		IF 前左轮力偏差 >200 THEN
			前左轮力偏差 := 200;
		END_IF
		IF 0< 前左轮力偏差 AND 前左轮力偏差 < 150 THEN
			前左轮力偏差 := 0;
		END_IF
		IF 前左轮力偏差 <-200 THEN
			前左轮力偏差 := -200;
		END_IF
		IF -170< 前左轮力偏差 AND 前左轮力偏差 < 0 THEN
			前左轮力偏差 := 0;
		END_IF
		
		IF 前右轮力偏差 >200 THEN
			前右轮力偏差 := 200;
		END_IF
		IF 前右轮力偏差 <-200 THEN
			前右轮力偏差 := -200;
		END_IF
		IF -170< 前右轮力偏差 AND 前右轮力偏差 < 0 THEN
			前右轮力偏差 := 0;
		END_IF
		IF 0< 前右轮力偏差 AND 前右轮力偏差 < 150 THEN
			前右轮力偏差 := 0;
		END_IF

		IF 后左轮力偏差 >200 THEN
			后左轮力偏差 := 200;
		END_IF
		IF 后左轮力偏差 <-200 THEN
			后左轮力偏差 := -200;
		END_IF
		IF -170< 后左轮力偏差 AND 后左轮力偏差 < 0 THEN
			后左轮力偏差 := 0;
		END_IF
		IF 0< 后左轮力偏差 AND 后左轮力偏差 < 150 THEN
			后左轮力偏差 := 0;
		END_IF
		
		IF 后右轮力偏差 >200 THEN
			后右轮力偏差 := 200;
		END_IF
		IF 后右轮力偏差 <-200 THEN
			后右轮力偏差 := -200;
		END_IF
		IF -170< 后右轮力偏差 AND 后右轮力偏差 < 0 THEN
			后右轮力偏差 := 0;
		END_IF
		IF 0< 后右轮力偏差 AND 后右轮力偏差 < 150 THEN
			后右轮力偏差 := 0;
		END_IF
		
		偏差值pitch := -目标值pitch + pitch角度滤波;
		偏差值roll := -目标值roll + roll角度滤波;
		
		PITCH := (pitch角度滤波 - v_pitch)/0.005;
		ROLL := (roll角度滤波 - v_roll)/0.005;

		//角速度滤波
		PITCH滤波 := B0 * PITCH + B1 * PITCH_x1 + B2 * PITCH_x2 - A1 * PITCH_y1 - A2 * PITCH_y2;
		PITCH_x2 := PITCH_x1;
		PITCH_x1 := PITCH;
		PITCH_y2 := PITCH_y1;
		PITCH_y1 := PITCH滤波;
		
		ROLL滤波 := B0 * ROLL + B1 * ROLL_x1 + B2 * ROLL_x2 - A1 * ROLL_y1 - A2 * ROLL_y2;
		ROLL_x2 := ROLL_x1;
		ROLL_x1 := ROLL;
		ROLL_y2 := ROLL_y1;
		ROLL_y1 := ROLL滤波;
		
// 死区处理
		IF ABS(偏差值pitch) < 误差死区 THEN 偏差值pitch := 0.0; END_IF;
		IF ABS(偏差值roll) < 误差死区 THEN 偏差值roll := 0.0; END_IF;
		
		IF ABS(偏差值pitch) < 误差死区 THEN PITCH滤波 := 0.0; END_IF;
		IF ABS(偏差值roll) < 误差死区 THEN ROLL滤波 := 0.0; END_IF;

		KP_roll := 0.45;
		KD_roll := 0.3;
		KI_roll := 0.0045;
		KP_pitch := 0.75;
		KD_pitch := 0.55;
		KI_pitch := 0.0045;

		//记录数据
		KD数据pitch := 偏差值pitch - 2*e_pitch_prev1 + e_pitch_prev2;
		KP数据pitch := 偏差值pitch - e_pitch_prev1;
		KI数据pitch := 偏差值pitch;
		KD数据roll := 偏差值roll - 2*e_roll_prev1 + e_roll_prev2;
		KP数据roll := 偏差值roll - e_roll_prev1;
		KI数据roll := 偏差值roll;
		
		// KP_pitch滤波计算
		KP数据pitch滤波 := B0 * KP数据pitch + B1 * KP_pitch_x1 + B2 * KP_pitch_x2 - A1 * KP_pitch_y1 - A2 * KP_pitch_y2;
		KP_pitch_x2 := KP_pitch_x1;
		KP_pitch_x1 := KP数据pitch;
		KP_pitch_y2 := KP_pitch_y1;
		KP_pitch_y1 := KP数据pitch滤波;
		
		KD数据pitch滤波 := B0 * KD数据pitch + B1 * KD_pitch_x1 + B2 * KD_pitch_x2 - A1 * KD_pitch_y1 - A2 * KD_pitch_y2;
		KD_pitch_x2 := KD_pitch_x1;
		KD_pitch_x1 := KD数据pitch;
		KD_pitch_y2 := KD_pitch_y1;
		KD_pitch_y1 := KD数据pitch滤波;
		
		KP数据roll滤波 := B0 * KP数据roll + B1 * KP_roll_x1 + B2 * KP_roll_x2 - A1 * KP_roll_y1 - A2 * KP_roll_y2;
		KP_roll_x2 := KP_roll_x1;
		KP_roll_x1 := KP数据roll;
		KP_roll_y2 := KP_roll_y1;
		KP_roll_y1 := KP数据roll滤波;

		KD数据roll滤波 := B0 * KD数据roll + B1 * KD_roll_x1 + B2 * KD_roll_x2 - A1 * KD_roll_y1 - A2 * KD_roll_y2;
		KD_roll_x2 := KD_roll_x1;
		KD_roll_x1 := KD数据roll;
		KD_roll_y2 := KD_roll_y1;
		KD_roll_y1 := KD数据roll滤波;

// PID输出
		控制量pitch := KP_pitch * (KP数据pitch滤波) 
            + KI_pitch * 偏差值pitch 
            + KD_pitch * (KD数据pitch滤波);
		
		控制量roll := KP_roll * (KP数据roll滤波) 
           + KI_roll * 偏差值roll 
           + KD_roll * (KD数据roll滤波);
		
		v_pitch := pitch角度滤波;
		v_roll := roll角度滤波;
		
		前左轮date_l := +控制量pitch - 控制量roll;
		前右轮date_l := +控制量pitch + 控制量roll;
		后左轮date_l := -控制量pitch - 控制量roll;
		后右轮date_l := -控制量pitch + 控制量roll;
		
		// 更新历史误差
		e_pitch_prev2 := e_pitch_prev1;
		e_pitch_prev1 := 偏差值pitch;
		e_roll_prev2 := e_roll_prev1;
		e_roll_prev1 := 偏差值roll;
        
		
		//弃用的力增益分段式		
		// 		IF ABS(前左轮力偏差)>180 THEN
		// 			KP_force前左 := 0.0012;
		// 			ELSE
		// 			KP_force前左 := 0.0006;
		// 		END_IF
		// 		
		// 		IF ABS(前右轮力偏差)>180 THEN
		// 			KP_force前右 := 0.0012;
		// 			ELSE
		// 			KP_force前右 := 0.0006;
		// 		END_IF
		// 
		// 		IF ABS(后左轮力偏差)>180 THEN
		// 			KP_force后左 := 0.0012;
		// 			ELSE
		// 			KP_force后左 := 0.0006;
		// 		END_IF
		// 
		// 		IF ABS(后右轮力偏差)>180 THEN
		// 			KP_force后右 := 0.0012;
		// 			ELSE
		// 			KP_force后右 := 0.0006;
		// 		END_IF

//调节力的增益与加速度
		// 前左轮速度滤波计算
		前左轮速度滤波 := B0 * 前左轮行驶速度 + B1 * FLa_x1 + B2 * FLa_x2 - A1 * FLa_y1 - A2 * FLa_y2;
		FLa_x2 := FLa_x1;
		FLa_x1 := 前左轮行驶速度;
		FLa_y2 := FLa_y1;
		FLa_y1 := 前左轮速度滤波;
		
		// 前右------------------------
		前右轮速度滤波 := B0 * 前右轮行驶速度 + B1 * FRa_x1 + B2 * FRa_x2 - A1 * FRa_y1 - A2 * FRa_y2;
		FRa_x2 := FRa_x1;
		FRa_x1 := 前右轮行驶速度;
		FRa_y2 := FRa_y1;
		FRa_y1 := 前右轮速度滤波;
		
		// 后左------------------------
		后左轮速度滤波 := B0 * 后左轮行驶速度 + B1 * RLa_x1 + B2 * RLa_x2 - A1 * RLa_y1 - A2 * RLa_y2;
		RLa_x2 := RLa_x1;
		RLa_x1 := 后左轮行驶速度;
		RLa_y2 := RLa_y1;
		RLa_y1 := 后左轮速度滤波;
		
		// 后右------------------------
		后右轮速度滤波 := B0 * 后右轮行驶速度 + B1 * RRa_x1 + B2 * RRa_x2 - A1 * RRa_y1 - A2 * RRa_y2;
		RRa_x2 := RRa_x1;
		RRa_x1 := 后右轮行驶速度;
		RRa_y2 := RRa_y1;
		RRa_y1 := 后右轮速度滤波;

        前左轮加速度滤波 := (前左轮速度滤波 - 前左轮速度滤波L)/0.005;
		前右轮加速度滤波 := (前右轮速度滤波 - 前右轮速度滤波L)/0.005;
		后左轮加速度滤波 := (后左轮速度滤波 - 后左轮速度滤波L)/0.005;
		后右轮加速度滤波 := (后右轮速度滤波 - 后右轮速度滤波L)/0.005;
		
		前左轮速度滤波L := 前左轮速度滤波;
		前右轮速度滤波L := 前右轮速度滤波;
		后左轮速度滤波L := 后左轮速度滤波;
		后右轮速度滤波L := 后右轮速度滤波;

// 弃用的定时器
		//accel_high := (ABS(后左轮加速度滤波) >= 150);
		//// 配置并运行定时器（预设时间50ms）
		//timer_high(IN:=accel_high, PT:=T#50MS);
		//IF timer_high.Q THEN
		//KP_force后左 :=  150*KP_force后左/ABS(后左轮加速度滤波) ;
		//KP_force前左 :=  150*KP_force前左/ABS(后左轮加速度滤波) ;
		//KP_force前右 :=  150*KP_force前右/ABS(后左轮加速度滤波) ;
		//KP_force后右 :=  150*KP_force后右/ABS(后左轮加速度滤波) ;
		//END_IF

		// 后左轮加速度计数器
		IF ABS(后左轮加速度滤波) >= 200 THEN
			a轮与kp力计数器 := a轮与kp力计数器 + 1;
		ELSE
			a轮与kp力计数器 := 0;
		END_IF;
		
		// 前左轮KP_force自适应调整
		IF ABS(前左轮力偏差) > 180 THEN
			KP_force前左 := KP_force前左 + 0.000011;
			IF KP_force前左 >= 0.0003 THEN
				KP_force前左 := 0.0003;
			END_IF;	
		ELSIF a轮与kp力计数器 >= 10 THEN
			KP_force前左 := KP_force前左 - 0.000011;
			IF KP_force前左 <= 0 THEN
				KP_force前左 := 0;
			END_IF;
		ELSIF a轮与kp力计数器 = 0 THEN
			IF KP_force前左 < 0.00015 THEN
				KP_force前左 := KP_force前左 + 0.000012;
			ELSIF KP_force前左 > 0.00015 THEN
				KP_force前左 := KP_force前左 - 0.000012;
			END_IF;
		END_IF;

		// 前右轮KP_force自适应调整
		IF ABS(前右轮力偏差) > 180 THEN
			KP_force前右 := KP_force前右 + 0.000011;
			IF KP_force前右 >= 0.0003 THEN
				KP_force前右 := 0.0003;
			END_IF;	
		ELSIF a轮与kp力计数器 >= 10 THEN
			KP_force前右 := KP_force前右 - 0.000011;
			IF KP_force前右 <= 0 THEN
				KP_force前右 := 0;
			END_IF;
		ELSIF a轮与kp力计数器 = 0 THEN
			IF KP_force前右 < 0.00015 THEN
				KP_force前右 := KP_force前右 + 0.000012;
			ELSIF KP_force前右 > 0.00015 THEN
				KP_force前右 := KP_force前右 - 0.000012;
			END_IF;
		END_IF;

		// 后左轮KP_force自适应调整
		IF ABS(后左轮力偏差) > 180 THEN
			KP_force后左 := KP_force后左 + 0.000012;
			IF KP_force后左 >= 0.0003 THEN
				KP_force后左 := 0.0003;
			END_IF;	
		ELSIF a轮与kp力计数器 >= 10 THEN
			KP_force后左 := KP_force后左 - 0.000012;
			IF KP_force后左 <= 0 THEN
				KP_force后左 := 0;
			END_IF;
		ELSIF a轮与kp力计数器 = 0 THEN
			IF KP_force后左 < 0.00015 THEN
				KP_force后左 := KP_force后左 + 0.000012;
			ELSIF KP_force后左 > 0.00015 THEN
				KP_force后左 := KP_force后左 - 0.000012;
			END_IF;
		END_IF;

		// 后右轮KP_force自适应调整
		IF ABS(后右轮力偏差) > 180 THEN
			KP_force后右 := KP_force后右 + 0.000012;
			IF KP_force后右 >= 0.0003 THEN
				KP_force后右 := 0.0003;
			END_IF;	
		ELSIF a轮与kp力计数器 >= 10 THEN
			KP_force后右 := KP_force后右 - 0.000012;
			IF KP_force后右 <= 0 THEN
				KP_force后右 := 0;
			END_IF;
		ELSIF a轮与kp力计数器 = 0 THEN
			IF KP_force后右 < 0.00015 THEN
				KP_force后右 := KP_force后右 + 0.000012;
			ELSIF KP_force后右 > 0.00015 THEN
				KP_force后右 := KP_force后右 - 0.000012;
			END_IF;
		END_IF;

		// 		IF ABS(后左轮加速度滤波) >= 200 THEN
		// 			KP_force后左 := 0;
		// 			KP_force前左 := 0;
		// 			KP_force前右 := 0;
		// 			KP_force后右 := 0;
		// 			ELSIF ABS(后左轮加速度滤波) >= 20 THEN
		// 			KP_force后左 :=  20*KP_force后左/ABS(后左轮加速度滤波) ;
		// 			KP_force前左 :=  20*KP_force前左/ABS(后左轮加速度滤波) ;
		// 			KP_force前右 :=  20*KP_force前右/ABS(后左轮加速度滤波) ;
		// 			KP_force后右 :=  20*KP_force后右/ABS(后左轮加速度滤波) ;
		// 		END_IF
		
		前左轮date := (前左轮date_l - (前左轮力偏差 * KP_force前左));
		前右轮date := (前右轮date_l - (前右轮力偏差 * KP_force前右));
		后左轮date := (后左轮date_l - (后左轮力偏差 * KP_force后左));
		后右轮date := (后右轮date_l - (后右轮力偏差 * KP_force后右));
		
		前左轮date_F := 前左轮力偏差 * KP_force前左;
		前右轮date_F := 前右轮力偏差 * KP_force前右;
		后左轮date_F := 后左轮力偏差 * KP_force后左;
		后右轮date_F := 后右轮力偏差 * KP_force后右;
		
		// 计算预期位置
		前左轮new := (前左轮输出 + 前左轮date);
		前右轮new := (前右轮输出 + 前右轮date);
		后左轮new := (后左轮输出 + 后左轮date);
		后右轮new := (后右轮输出 + 后右轮date);
		
//执行器极限补偿
		//前轮组极限检查
		前轮组上极限 := (前左轮new >= 执行器行程限制) AND (前右轮new >= 执行器行程限制);
		前轮组下极限 := (前左轮new <= -执行器行程限制) AND (前右轮new <= -执行器行程限制);
		
		// 后轮组极限检查
		后轮组上极限 := (后左轮new >= 执行器行程限制) AND (后右轮new >= 执行器行程限制);
		后轮组下极限 := (后左轮new <= -执行器行程限制) AND (后右轮new <= -执行器行程限制);
		
		// Pitch轴补偿
		IF 前轮组上极限 AND (偏差值pitch > 误差死区) THEN
			后左轮date := 后左轮date - 最大调整速度 * 0.01;
			后右轮date := 后右轮date - 最大调整速度 * 0.01;
		ELSIF 前轮组下极限 AND (偏差值pitch < -误差死区) THEN
			后左轮date := 后左轮date + 最大调整速度 * 0.01;
			后右轮date := 后右轮date + 最大调整速度 * 0.01;
		END_IF;
		
		IF 后轮组上极限 AND (偏差值pitch < -误差死区) THEN
			前左轮date := 前左轮date + 最大调整速度 * 0.01;
			前右轮date := 前右轮date + 最大调整速度 * 0.01;
		ELSIF 后轮组下极限 AND (偏差值pitch > 误差死区) THEN
			前左轮date := 前左轮date - 最大调整速度 * 0.01;
			前右轮date := 前右轮date - 最大调整速度 * 0.01;
		END_IF;
		
		// 左侧极限检查
		左组轮上极限 := (前左轮new >= 执行器行程限制) AND (后左轮new >= 执行器行程限制);
		左组轮下极限 := (前左轮new <= -执行器行程限制) AND (后左轮new <= -执行器行程限制);
		
		// 右侧极限检查
		右组轮上极限 := (前右轮date >= 执行器行程限制) AND (后右轮date >= 执行器行程限制);
		右组轮下极限 := (前右轮date <= -执行器行程限制) AND (后右轮date <= -执行器行程限制);
		
		IF 左组轮上极限 AND (偏差值roll > 误差死区) THEN
			前右轮date := 前右轮date - 最大调整速度 * 0.01;
			后右轮date := 后右轮date - 最大调整速度 * 0.01;
		ELSIF 左组轮下极限 AND (偏差值roll < -误差死区) THEN
			前右轮date := 前右轮date + 最大调整速度 * 0.01;
			后右轮date := 后右轮date + 最大调整速度 * 0.01;
		END_IF;
		
		IF 右组轮上极限 AND (偏差值roll < -误差死区) THEN
			前左轮date := 前左轮date - 最大调整速度 * 0.01;
			后左轮date := 后左轮date - 最大调整速度 * 0.01;
		ELSIF 右组轮下极限 AND (偏差值roll > 误差死区) THEN
			前左轮date := 前左轮date + 最大调整速度 * 0.01;
			后左轮date := 后左轮date + 最大调整速度 * 0.01;
		END_IF;
		
		//最终限幅及输出
		// 速度限幅
		前左轮date := LIMIT(前左轮date, -最大调整速度, 最大调整速度);
		前右轮date := LIMIT(前右轮date, -最大调整速度, 最大调整速度);
		后左轮date := LIMIT(后左轮date, -最大调整速度, 最大调整速度);
		后右轮date := LIMIT(后右轮date, -最大调整速度, 最大调整速度);

//弃用的速度控制
		// 前左轮速度计算
		IF ABS(前左轮date) > 10.0 THEN
			前左轮速度 := 50.0;
		ELSIF ABS(前左轮date) < 0.05 THEN
			前左轮速度 := 0.0;
		ELSE
			前左轮速度 := (前左轮date) * (50.0 / 10);  // 100/(10.0-0.5)=10.5263
		END_IF;
		
		// 前右轮速度计算
		IF ABS(前右轮date) > 10.0 THEN
			前右轮速度 := 50.0;
		ELSIF ABS(前右轮date) < 0.05 THEN
			前右轮速度 := 0.0;
		ELSE
			前右轮速度 := (前右轮date) * (50.0 / 10);
		END_IF;
		
		// 后左轮速度计算
		IF ABS(后左轮date) > 10.0 THEN
			后左轮速度 := 50.0;
		ELSIF ABS(后左轮date) < 0.05 THEN
			后左轮速度 := 0.0;
		ELSE
			后左轮速度 := (后左轮date) * (50.0 / 10);
		END_IF;
		
		// 后右轮速度计算
		IF ABS(后右轮date) > 10.0 THEN
			后右轮速度 := 50.0;
		ELSIF ABS(后右轮date) < 0.05 THEN
			后右轮速度 := 0.0;
		ELSE
			后右轮速度 := (后右轮date) * (50.0 / 10);
		END_IF;
		
		delta前左 := 前左轮date - 前左轮date_l_prev;
		delta前右 := 前右轮date - 前右轮date_l_prev;
		delta后左 := 后左轮date - 后左轮date_l_prev;
		delta后右 := 后右轮date - 后右轮date_l_prev;
		
		//前左轮date_prev := 前左轮date;
		//前右轮date_prev := 前右轮date;
		//后左轮date_prev := 后左轮date;
		//后右轮date_prev := 后右轮date;

//轮date增幅限制
		//前左
		IF delta前左 > 0 THEN
			sign := 1;      // 正方向
		ELSIF delta前左 < 0 THEN
			sign := -1;     // 负方向
		ELSE
			sign := 0;      // 无变化
		END_IF;
		
		IF ABS(delta前左) > delta_threshold THEN
			// 超过阈值时，按符号限幅
			前左轮date := 前左轮date_l_prev + (sign * delta_threshold);
		END_IF;
		//前右
		IF delta前右 > 0 THEN
			sign := 1;      // 正方向
		ELSIF delta前右 < 0 THEN
			sign := -1;     // 负方向
		ELSE
			sign := 0;      // 无变化
		END_IF;
		
		IF ABS(delta前右) > delta_threshold THEN
			// 超过阈值时，按符号限幅
			前右轮date := 前右轮date_l_prev + (sign * delta_threshold);
		END_IF;
        //后左
		IF delta后左 > 0 THEN
			sign := 1;      // 正方向
		ELSIF delta后左 < 0 THEN
			sign := -1;     // 负方向
		ELSE
			sign := 0;      // 无变化
		END_IF;
		
		IF ABS(delta后左) > delta_threshold THEN
			// 超过阈值时，按符号限幅
			后左轮date := 后左轮date_l_prev + (sign * delta_threshold);
		END_IF;
		//后右
		IF delta后右 > 0 THEN
			sign := 1;      // 正方向
		ELSIF delta后右 < 0 THEN
			sign := -1;     // 负方向
		ELSE
			sign := 0;      // 无变化
		END_IF;
		
		IF ABS(delta后右) > delta_threshold THEN
			// 超过阈值时，按符号限幅
			后右轮date := 后右轮date_l_prev + (sign * delta_threshold);
		END_IF;

		前左轮date_l_prev := 前左轮date;
		前右轮date_l_prev := 前右轮date;
		后右轮date_l_prev := 后右轮date;
		后左轮date_l_prev := 后左轮date;

//轮date滤波
		// 前左轮滤波计算
		// ----------------------------
		前左轮date滤波 := B0 * 前左轮date + B1 * FLdate_x1 + B2 * FLdate_x2 - A1 * FLdate_y1 - A2 * FLdate_y2;
		// 更新状态
		FLdate_x2 := FLdate_x1;
		FLdate_x1 := 前左轮date;
		FLdate_y2 := FLdate_y1;
		FLdate_y1 := 前左轮date滤波;
		
		// ----------------------------
		// 前右轮滤波计算
		// ----------------------------
		前右轮date滤波 := B0 * 前右轮date + B1 * FRdate_x1 + B2 * FRdate_x2 - A1 * FRdate_y1 - A2 * FRdate_y2;
		// 更新状态
		FRdate_x2 := FRdate_x1;
		FRdate_x1 := 前右轮date;
		FRdate_y2 := FRdate_y1;
		FRdate_y1 := 前右轮date滤波;
		
		// ----------------------------
		// 后左轮滤波计算
		// ----------------------------
		后左轮date滤波 := B0 * 后左轮date + B1 * BLdate_x1 + B2 * BLdate_x2 - A1 * BLdate_y1 - A2 * BLdate_y2;
		// 更新状态
		BLdate_x2 := BLdate_x1;
		BLdate_x1 := 后左轮date;
		BLdate_y2 := BLdate_y1;
		BLdate_y1 := 后左轮date滤波;
		
		// ----------------------------
		// 后右轮滤波计算
		// ----------------------------
		后右轮date滤波 := B0 * 后右轮date + B1 * BRdate_x1 + B2 * BRdate_x2 - A1 * BRdate_y1 - A2 * BRdate_y2;
		// 更新状态
		BRdate_x2 := BRdate_x1;
		BRdate_x1 := 后右轮date;
		BRdate_y2 := BRdate_y1;
		BRdate_y1 := 后右轮date滤波;

// 前左轮date滤波应用限幅（±0.01米）
		// 前左轮date滤波 := LIMIT(前左轮date滤波, -0.25, 0.25);
		// 前右轮date滤波 := LIMIT(前右轮date滤波, -0.25, 0.25);
		// 后左轮date滤波 := LIMIT(后左轮date滤波, -0.25, 0.25);
		// 后右轮date滤波 := LIMIT(后右轮date滤波, -0.25, 0.25);

		平均实际长度 := (前左轮实际长度 + 前右轮实际长度 + 后左轮实际长度 + 后右轮实际长度) / 4.0;

		IF 平均实际长度>0.5 AND ABS(pitch角度滤波) < 0.5 AND ABS(roll角度滤波) < 0.5 THEN
			// 模式A：偏差均小时，用比例调整输出
			前左轮输出 := LIMIT(前左轮输出 + 前左轮date滤波 + 前左轮调整量滤波 - kp * 15, -执行器行程限制, 执行器行程限制);
			前右轮输出 := LIMIT(前右轮输出 + 前右轮date滤波 + 前右轮调整量滤波 - kp * 15, -执行器行程限制, 执行器行程限制);
			后左轮输出 := LIMIT(后左轮输出 + 后左轮date滤波 + 后左轮调整量滤波 - kp * 15, -执行器行程限制, 执行器行程限制);
			后右轮输出 := LIMIT(后右轮实际长度 + 后右轮date滤波 + 后右轮调整量滤波 - kp * 15, -执行器行程限制, 执行器行程限制);
			ELSE IF 平均实际长度<-0.5 AND ABS(pitch角度滤波) < 0.5 AND ABS(roll角度滤波) < 0.5 THEN
			前左轮输出 := LIMIT(前左轮输出 + 前左轮date滤波 + 前左轮调整量滤波 + kp * 15, -执行器行程限制, 执行器行程限制);
			前右轮输出 := LIMIT(前右轮输出 + 前右轮date滤波 + 前右轮调整量滤波 + kp * 15, -执行器行程限制, 执行器行程限制);
			后左轮输出 := LIMIT(后左轮输出 + 后左轮date滤波 + 后左轮调整量滤波 + kp * 15, -执行器行程限制, 执行器行程限制);
			后右轮输出 := LIMIT(后右轮输出 + 后右轮date滤波 + 后右轮调整量滤波 + kp * 15, -执行器行程限制, 执行器行程限制);
					ELSE
						前左轮输出 := LIMIT(前左轮输出 + 前左轮date滤波 + 前左轮调整量滤波, -执行器行程限制, 执行器行程限制);
						前右轮输出 := LIMIT(前右轮输出 + 前右轮date滤波 + 前右轮调整量滤波, -执行器行程限制, 执行器行程限制);
						后左轮输出 := LIMIT(后左轮输出 + 后左轮date滤波 + 后左轮调整量滤波, -执行器行程限制, 执行器行程限制);
						后右轮输出 := LIMIT(后右轮输出 + 后右轮date滤波 + 后右轮调整量滤波, -执行器行程限制, 执行器行程限制);
			     END_IF
		END_IF;

END_FUNCTION_BLOCK

// Device/Application/函数/运动控制/伺服控制
FUNCTION_BLOCK 伺服控制
VAR_INPUT
	pAxis      	: POINTER TO AXIS_REF_SM3;	//定义轴
END_VAR
VAR_OUTPUT
END_VAR
VAR
	前进					: BOOL := FALSE;
	后退					: BOOL := FALSE;
	运动到点开始,运动到点开始1			: BOOL := FALSE;
	相对运动到点开始        : BOOL := FALSE;
	连续运动到点开始        : BOOL := FALSE;
	速度运动到点开始,速度运动到点开始1        : BOOL := FALSE;
	力矩模式切换: BOOL;
	力矩控制,力矩控制1:BOOL;
	暂停        : BOOL := FALSE;
	停止控制    : BOOL := FALSE;
	
	到点位置				: LREAL := 0.0;
	pMC_Jog    			: MC_Jog;
	pMC_Power  			: MC_Power;
	pMC_Reset  			: MC_Reset;
	pMC_MoveAbsolute1,pMC_MoveAbsolute 	: MC_MoveAbsolute;
	pMC_MoveRelative 	: MC_MoveRelative;
	pMC_MoveAdditive    : MC_MoveAdditive;
	pMC_MoveVelocity,pMC_MoveVelocity1    : MC_MoveVelocity;
	pSMC_SetTorque,pSMC_SetTorque1      : SMC_SetTorque;
	pSMC_MoveContinuousAbsolute: SMC_MoveContinuousAbsolute;
	pSMC_SetControllerMode:SMC_SetControllerMode;
	pMC_Halt:MC_Halt;
	pMC_Stop:MC_Stop;
	pSMC3_ReinitDrive:SMC3_ReinitDrive;
	运行速度		: LREAL ;
	运行方向		: INT ;
	
END_VAR
VAR_IN_OUT
	伺服参数    			: 伺服参数结构体;
END_VAR

IF 轴报警=FALSE THEN
CASE 伺服参数.运行模式 OF
	0 :	// 无运动
		前进 := FALSE;
		后退 := FALSE;
		运动到点开始:=FALSE;
		运动到点开始1:=FALSE;
		相对运动到点开始:=FALSE;
		连续运动到点开始:=FALSE;
		速度运动到点开始:=FALSE;
		速度运动到点开始1:=FALSE;
		力矩控制:=FALSE;
		力矩控制1:=FALSE;
		暂停:=FALSE;
		停止控制:=FALSE;
		力矩模式切换:=FALSE;
		//轴复位:=FALSE;
		//轴初始化:=FALSE;
	1 : // 点动运行
		IF 伺服参数.运行方向=TRUE THEN
			前进 := TRUE;
			后退 := FALSE;
		ELSE
			前进 := FALSE;
			后退 := TRUE;
		END_IF
	2 : // 运动到点1
	    运动到点开始1:=FALSE;
		运动到点开始:=TRUE;
	3 : // 相对运动
	    运动到点开始:=FALSE;
		运动到点开始1:=FALSE;
		相对运动到点开始:=TRUE;
		
	4 : // 运动到点2
	    运动到点开始:=FALSE;
		运动到点开始1:=TRUE;
	
    5:
	    暂停:=TRUE;
	6://速度控制1
	    速度运动到点开始1:=FALSE;
	    速度运动到点开始:=TRUE;
		暂停:=FALSE;
	7://速度控制2
	    速度运动到点开始:=FALSE;
	    速度运动到点开始1:=TRUE;
		暂停:=FALSE;
	8://力矩控制1
	    力矩控制1:=FALSE;
		力矩控制:=TRUE;
	9://力矩控制2
	    力矩控制:=FALSE;
		力矩控制1:=TRUE;
	10://停止
	    停止控制:=TRUE;
	11://力矩切换
	    力矩模式切换:=TRUE;
	//12://位置模式
	(*
	13://复位
	    轴复位:=TRUE;
	14://初始化
	    轴初始化:=TRUE;
	*)
END_CASE
END_IF
pMC_Power(
	Axis:= pAxis^,
	Enable:= TRUE,
	bRegulatorOn:= 伺服参数.使能,
	bDriveStart:= TRUE,
	Status=> , 
	bRegulatorRealState=> 伺服参数.使能状态.DONE, 
	bDriveStartRealState=> , 
	Busy=> 伺服参数.使能状态.BUSY, 
	Error=> 伺服参数.使能状态.Error, 
	ErrorID=> 伺服参数.使能状态.ErrorID);

pMC_Jog(
	Axis:= pAxis^,
	JogForward:= 前进,
	JogBackward:= 后退,
	Velocity:= 伺服参数.运行速度,
	Acceleration:= 10000,
	Deceleration:= 10000,
	Jerk:=100000,
	Busy=> 伺服参数.点动运行中,
	CommandAborted=>,
	Error=>, 
	ErrorId=> );

pMC_MoveAbsolute(
	Axis:=pAxis^ , 
	Execute:= 运动到点开始, 
	Position:= 伺服参数.运行位置, 
	Velocity:= 伺服参数.运行速度, 
	Acceleration:= 10000, 
	Deceleration:= 10000, 
	Jerk:= 100000, 
	Direction:= , 
	BufferMode:= 0, 
	Done=> 伺服参数.绝对定位状态.DONE, 
	Busy=> 伺服参数.绝对定位状态.BUSY, 
	CommandAborted=> 伺服参数.绝对定位状态.CommandAborted, 
	Error=> 伺服参数.绝对定位状态.Error, 
	ErrorID=> 伺服参数.绝对定位状态.ErrorID);	

pMC_MoveAbsolute1(
	Axis:=pAxis^ , 
	Execute:= 运动到点开始1, 
	Position:= 伺服参数.运行位置1, 
	Velocity:= 伺服参数.运行速度, 
	Acceleration:= 10000, 
	Deceleration:= 10000, 
	Jerk:= 100000, 
	Direction:= , 
	BufferMode:= 0, 
	Done=> 伺服参数.绝对定位状态1.DONE, 
	Busy=> 伺服参数.绝对定位状态1.BUSY, 
	CommandAborted=> 伺服参数.绝对定位状态1.CommandAborted, 
	Error=> 伺服参数.绝对定位状态1.Error, 
	ErrorID=> 伺服参数.绝对定位状态1.ErrorID);	

pMC_MoveRelative(
	Axis:= pAxis^, 
	Execute:= 相对运动到点开始, 
	Distance:= 伺服参数.运行位置, 
	Velocity:= 伺服参数.运行速度, 
	Acceleration:= 500, 
	Deceleration:= 500, 
	Jerk:= 5000, 
	BufferMode:= 5, 
	Done=> 伺服参数.相对定位状态.DONE, 
	Busy=> 伺服参数.相对定位状态.BUSY, 
	Active=> , 
	CommandAborted=> 伺服参数.相对定位状态.CommandAborted, 
	Error=> 伺服参数.相对定位状态.Error, 
	ErrorID=> 伺服参数.相对定位状态.ErrorID);
(*
pMC_MoveAdditive(
	Axis:= pAxis^, 
	Execute:= 运动到点开始1, 
	Distance:= 伺服参数.运行位置1, 
	Velocity:= 伺服参数.运行速度, 
	Acceleration:= 5000, 
	Deceleration:= 5000, 
	Jerk:= 50000, 
	Done=> 伺服参数.运动到点完成1, 
	Busy=> , 
	CommandAborted=> , 
	Error=> , 
	ErrorID=> );
*)
(*
pSMC_MoveContinuousAbsolute(
	Axis:= pAxis^, 
	Execute:= 连续运动到点开始, 
	Position:= 伺服参数.运行位置, 
	Velocity:= 伺服参数.运行速度, 
	EndVelocity:=伺服参数.结束运行速度, 
	EndVelocityDirection:= , 
	Acceleration:= 500, 
	Deceleration:= 500, 
	Jerk:= 5000, 
	Direction:= , 
	AdaptEndVelToAvoidOvershoot:=TRUE,
	InEndVelocity=> , 
	PositionReached=> 伺服参数.连续运动到点完成, 
	Busy=> , 
	CommandAborted=> , 
	Error=> , 
	ErrorID=> );
*)
pMC_Halt(
	Axis:= pAxis^, 
	Execute:= 暂停, 
	Deceleration:= 500, 
	Jerk:= 5000, 
	Done=> 伺服参数.暂停状态.DONE, 
	Busy=> 伺服参数.暂停状态.BUSY, 
	CommandAborted=> 伺服参数.暂停状态.CommandAborted, 
	Error=> 伺服参数.暂停状态.Error, 
	ErrorID=> 伺服参数.暂停状态.ErrorID);
	
pMC_Reset(
	Axis:= pAxis^, 
	Execute:= 伺服参数.轴复位, 
	Done=> 伺服参数.复位状态.DONE, 
	Busy=> 伺服参数.复位状态.BUSY, 
	Error=> 伺服参数.复位状态.Error, 
	ErrorID=> 伺服参数.复位状态.ErrorID);
pSMC3_ReinitDrive(
	Axis:= pAxis^, 
	bExecute:= 伺服参数.轴初始化, 
	bVirtual:= , 
	bDone=> 伺服参数.初始化状态.DONE, 
	bBusy=> 伺服参数.初始化状态.BUSY, 
	bError=> 伺服参数.初始化状态.Error, 
	nErrorID=> 伺服参数.初始化状态.ErrorID);


////////////////////////////////////////////////////////////////////////////////////////////////////////

pMC_MoveVelocity(
	Axis:= pAxis^, 
	Execute:= 速度运动到点开始 , 
	Velocity:= 伺服参数.运行控制速度, 
	Acceleration:= 200, 
	Deceleration:= 300, 
	Jerk:= 200, 
	Direction:= 伺服参数.运行控制方向, 
	BufferMode:= , 
	InVelocity=> 伺服参数.速度运动状态.DONE, 
	Busy=> 伺服参数.速度运动状态.BUSY, 
	Active=> , 
	CommandAborted=> 伺服参数.速度运动状态.CommandAborted, 
	Error=> 伺服参数.速度运动状态.Error, 
	ErrorID=> 伺服参数.速度运动状态.ErrorID);
	
pMC_MoveVelocity1(
	Axis:= pAxis^, 
	Execute:= 速度运动到点开始1 , 
	Velocity:= 伺服参数.运行控制速度1, 
	Acceleration:= 200, 
	Deceleration:= 300, 
	Jerk:= 200, 
	Direction:= 伺服参数.运行控制方向, 
	BufferMode:= , 
	InVelocity=> 伺服参数.速度运动状态1.DONE, 
	Busy=> 伺服参数.速度运动状态1.BUSY, 
	Active=> , 
	CommandAborted=> 伺服参数.速度运动状态1.CommandAborted, 
	Error=> 伺服参数.速度运动状态1.Error, 
	ErrorID=> 伺服参数.速度运动状态1.ErrorID);
//轴程序控制.伺服反馈_速度运行_done := 速度运动状态.DONE;	

pSMC_SetControllerMode(
	Axis:= pAxis^, 
	bExecute:= 力矩模式切换 AND NOT (pAxis^.nAxisState = 1 OR pAxis^.nAxisState = 2 OR pAxis^.nAxisState = 7), 
	nControllerMode:= 伺服参数.控制模式, 
	bDone=> 伺服参数.控制模式切换状态.DONE, 
	bBusy=> 伺服参数.控制模式切换状态.BUSY, 
	bError=> 伺服参数.控制模式切换状态.Error, 
	nErrorID=> 伺服参数.控制模式切换状态.ErrorID);
//伺服参数.控制模式切换完成 := pSMC_SetControllerMode.bDone; 



pSMC_SetTorque(
	Axis:=pAxis^ ,
	bEnable:=力矩控制 AND 伺服参数.控制模式 = SMC_torque  ,
	fTorque:=伺服参数.设定力矩 ,
    bBusy => , 
    bError => , 
    nErrorID => , 
	bBusy=> );
	
pSMC_SetTorque1(
	Axis:=pAxis^ ,
	bEnable:=力矩控制1 AND 伺服参数.控制模式 = SMC_torque  ,
	fTorque:=伺服参数.设定力矩1 ,
    bBusy => , 
    bError => , 
    nErrorID => , 
	bBusy=> );
//轴程序控制.伺服反馈_力矩运行_done := 力矩运动状态.BUSY;

pMC_Stop(
	Axis:= pAxis^, 
	Execute:= 伺服参数.停止控制, 
	Deceleration:= 2000, 
	Jerk:= 20000, 
	Done=> 伺服参数.停止状态.DONE, 
	Busy=> 伺服参数.停止状态.BUSY, 
	Error=> 伺服参数.停止状态.Error, 
	ErrorID=> 伺服参数.停止状态.ErrorID);
//轴程序控制.伺服反馈_停止_done := 停止状态.DONE;




伺服参数.指令位置 := pAxis^.fSetPosition;
伺服参数.指令力矩 := pAxis^.fSetTorque;
伺服参数.指令速度 := pAxis^.fSetVelocity;
伺服参数.反馈位置 := pAxis^.fActPosition;
伺服参数.反馈力矩 := pAxis^.fActTorque;
伺服参数.反馈速度 := pAxis^.fActVelocity;
伺服参数.反馈电流 := pAxis^.fActCurrent;
伺服参数.反馈状态 := pAxis^.nAxisState;

END_FUNCTION_BLOCK

// Device/Application/末端控制
PROGRAM 末端控制
VAR
	末端碰撞调整开关	: BOOL := FALSE;
	末端速度			: LREAL := 100.0;
	伸缩轴伺服控制    : 伺服控制;
	上卷扬伺服控制    : 伺服控制;
	下卷扬伺服控制    : 伺服控制;
	滚刷伺服控制    	: 伺服控制;
	
	// 滤波参数
	滤波系数			: LREAL := 0.1;
	上卷扬滤波力矩	: LREAL;
	下卷扬滤波力矩	: LREAL;
	上卷扬上周期力矩	: LREAL;
	下卷扬上周期力矩	: LREAL;
	上卷扬力矩限制	: LREAL := -30.0;
	下卷扬力矩限制	: LREAL := -30.0;
	
	上下卷扬速度系数:INT:=1;
	实时检测延时:TON;
	延时时间:TIME:=T#2S;
// 	bFirstRun		: BOOL := TRUE;
// 	bAutoControl	: BOOL := FALSE;
// 	iCounter		: INT := 0;
// 	iAxisNum		: INT := 0;
// 	bMoveStatus		: INT := 2;
// 	iVel			: INT := 2;
// 	
// 	adFbPos     	: ARRAY[0..3] OF LREAL;
	adFbForce    	: ARRAY[0..3] OF INT;
// 	abMC_Jog_Busy   : ARRAY[0..3] OF BOOL;
// 	abForward		: ARRAY[0..3] OF BOOL := [FALSE, FALSE, FALSE, FALSE];
// 	abBackward		: ARRAY[0..3] OF BOOL := [FALSE, FALSE, FALSE, FALSE];
// 	
// 	// 滤波参数
// 	dFilterFac		: LREAL := 0.3;
// 	adFbFilterForce	: ARRAY[0..3] OF LREAL;
// 	adFbLastForce	: ARRAY[0..3] OF LREAL;
// 	adForceLimit	: ARRAY[0..3] OF LREAL := [0.0, -150.0, -450.0, 0.0];
// 	
// 	apMC_Jog    	: ARRAY[0..3] OF MC_Jog;
// 	apMC_Power  	: ARRAY[0..3] OF MC_Power;
// 	apAxis      	: ARRAY[0..3] OF POINTER TO AXIS_REF_SM3;//定义轴


    卷扬1处理数值: REAL;
	卷扬2处理数值: REAL;
	PID_1: PID;
	PID_2: PID;
	卷扬1到位: BOOL;
	卷扬2到位: BOOL;
	卷扬1PID复位: BOOL;
	卷扬2PID复位: BOOL;
END_VAR

//ACT_test();
IF 末端使能=TRUE THEN
	伸缩轴伺服参数.使能 := TRUE;
	上卷扬伺服参数.使能 := TRUE;
	下卷扬伺服参数.使能 := TRUE;
	滚刷伺服参数.使能 := TRUE;
	伸缩轴伺服参数.运行速度 := 末端速度;
	上卷扬伺服参数.运行速度 := 末端速度*上下卷扬速度系数;
	下卷扬伺服参数.运行速度 := 末端速度*上下卷扬速度系数;
	滚刷伺服参数.运行速度 := 末端速度/7.0;
	IF 伸缩轴伺服参数.使能状态.DONE=TRUE THEN
		伸缩架使能完成:=TRUE;
	ELSE
	    伸缩架使能完成:=FALSE;
	END_IF
	IF 上卷扬伺服参数.使能状态.DONE=TRUE THEN
		上卷扬使能完成:=TRUE;
	ELSE
	    上卷扬使能完成:=FALSE;
	END_IF
	IF 下卷扬伺服参数.使能状态.DONE=TRUE THEN
		下卷扬使能完成:=TRUE;
	ELSE
	    下卷扬使能完成:=FALSE;
	END_IF
	IF 滚刷伺服参数.使能状态.DONE=TRUE THEN
		滚刷使能完成:=TRUE;
	ELSE
	    滚刷使能完成:=FALSE;
	END_IF
ELSE
	伸缩轴伺服参数.使能 := FALSE;
	上卷扬伺服参数.使能 := FALSE;
	下卷扬伺服参数.使能 := FALSE;
	滚刷伺服参数.使能 := FALSE;
END_IF

伸缩轴伺服控制(伺服参数:=伸缩轴伺服参数, pAxis:=ADR(伸缩轴));
上卷扬伺服控制(伺服参数:=上卷扬伺服参数, pAxis:=ADR(上卷扬));
下卷扬伺服控制(伺服参数:=下卷扬伺服参数, pAxis:=ADR(下卷扬));
滚刷伺服控制(伺服参数:=滚刷伺服参数, pAxis:=ADR(滚刷));
//上测力矩低通滤波模块(输入数据:= adFbForce[1], 滤波系数:= 滤波系数, 输出数据=>上卷扬滤波力矩 );
//下测力矩低通滤波模块(输入数据:= adFbForce[2], 滤波系数:= 滤波系数, 输出数据=>下卷扬滤波力矩 );
(*
上测力矩低通滤波模块(输入数据:= adFbForce[1], 滤波系数:= 滤波系数, 输出数据=>上卷扬滤波力矩 );
下测力矩低通滤波模块(输入数据:= adFbForce[2], 滤波系数:= 滤波系数, 输出数据=>下卷扬滤波力矩 );
IF 末端碰撞调整开关 = TRUE THEN
	IF 上卷扬滤波力矩 > 上卷扬力矩限制 THEN
		上卷扬伺服参数.运行模式 := 1;
		上卷扬伺服参数.运行方向 := FALSE;
	ELSE
		上卷扬伺服参数.运行模式 := 0;
	END_IF
	IF 下卷扬滤波力矩 > 下卷扬力矩限制 THEN
		下卷扬伺服参数.运行模式 := 1;
		下卷扬伺服参数.运行方向 := FALSE;
	ELSE
		下卷扬伺服参数.运行模式 := 0;
	END_IF
END_IF
*)
(*
上卷扬滤波力矩 := (1 - 滤波系数)*上卷扬上周期力矩 + 滤波系数*adFbForce[1];
上卷扬上周期力矩 := 上卷扬滤波力矩;

下卷扬滤波力矩 := (1 - 滤波系数)*下卷扬上周期力矩 + 滤波系数*adFbForce[2];
下卷扬上周期力矩 := 下卷扬滤波力矩;

IF 末端碰撞调整开关 = TRUE THEN
	IF 上卷扬滤波力矩 > 上卷扬力矩限制 THEN
		下卷扬伺服参数.运行模式 := 1;
		上卷扬伺服参数.运行方向 := FALSE;
	ELSIF 下卷扬滤波力矩 > 下卷扬力矩限制 THEN
		下卷扬伺服参数.运行模式 := 1;
		下卷扬伺服参数.运行方向 := FALSE;
	ELSE
		下卷扬伺服参数.运行模式 := 0;
	END_IF
END_IF
*)
CASE 控制方式 OF
	0 :	//手动控制
		回零控制();
	1 :	//自动控制
		传感器检测();
		上下卷扬控制();
		对中机构控制();
		回零控制();
		
		IF 上装自动运行 THEN
			CASE 上装自动流程 OF
			0:
			   对中机构自动流程:=0;
			   上下卷扬自动流程:=0;
			   启动对中机构自动运行:=FALSE;
			   启动上下扬自动运行:=FALSE;
			   对中工作完成:=FALSE;
			   上下卷扬工作完成:=FALSE;
			   上装自动流程:=10;
			10:
			   启动对中机构自动运行:=TRUE;
			   IF 对中工作完成 THEN
				   上装自动流程:=20;
			   END_IF
			20:
			   启动上下扬自动运行:=TRUE;
			   IF 上下卷扬工作完成 THEN
				   上装自动流程:=30;
			   END_IF
			30:
			   ;
			END_CASE
		END_IF
END_CASE

ACTION 上下卷扬控制:
IF 启动上下扬自动运行 THEN
CASE 上下卷扬自动流程 OF
	0:
	   上下卷扬检测数据有误:=FALSE;
	   上卷扬到达清扫面:=FALSE;
	   下卷扬到达清扫面:=FALSE;
	   上下卷扬工作完成:=FALSE;
	   上下卷扬自动流程:=5;
	   上下卷扬异常:=FALSE;
	   上卷扬伺服参数.运行模式:=0;
	   下卷扬伺服参数.运行模式:=0;
	   上卷扬伺服参数.绝对定位状态.DONE:=FALSE;
	   下卷扬伺服参数.绝对定位状态.DONE:=FALSE;
	   实时检测延时(IN:= FALSE, PT:= 延时时间, Q=> , ET=> );
	   卷扬1PID复位:=1;
	   卷扬2PID复位:=1;
	5:
	   IF 边沿检测1=1000 AND 边沿检测2=1000 AND 边沿检测3=1000 AND 边沿检测4=1000 
		   AND 超声波检测左1=1000 AND 超声波检测左2=1000 AND 超声波检测右1=1000 AND 超声波检测右2=1000 THEN
		   上卷扬伺服参数.运行位置:=26;
		   下卷扬伺服参数.运行位置:=20;
		   上卷扬伺服参数.运行模式:=3;
		   下卷扬伺服参数.运行模式:=3;
		   上下卷扬自动流程:=6;
	   ELSE
		   上下卷扬检测数据有误:=0;
		   上下卷扬自动流程:=10;
	   END_IF
	6:
	   IF 上卷扬伺服参数.相对定位状态.DONE OR 下卷扬伺服参数.相对定位状态.DONE THEN
		   上卷扬伺服参数.运行模式:=0;
		   下卷扬伺服参数.运行模式:=0;
		   IF 边沿检测1=1000 AND 边沿检测2=1000 AND 边沿检测3=1000 AND 边沿检测4=1000 
		   AND 超声波检测左1=1000 AND 超声波检测左2=1000 AND 超声波检测右1=1000 AND 超声波检测右2=1000 THEN
		      上下卷扬检测数据有误:=1;
		      上下卷扬自动流程:=1000;
	       ELSE
		      上下卷扬检测数据有误:=0;
		      上下卷扬自动流程:=10;
		   END_IF
	   END_IF
	10:
	   IF (边沿检测1<>1000 OR 边沿检测2<>1000) AND (边沿检测3=1000 OR 边沿检测4=1000) THEN
	   	   上下卷扬自动流程:=20;
	   ELSIF (边沿检测1=1000 OR 边沿检测2=1000) AND (边沿检测3<>1000 OR 边沿检测4<>1000) THEN
	   	   上下卷扬自动流程:=30;
	   ELSIF 边沿检测1=1000 AND 边沿检测2=1000 AND 边沿检测3=1000 AND 边沿检测4=1000 THEN
	   	   上下卷扬自动流程:=40;
	   END_IF
	30:
	   启动对中机构自动运行:=TRUE;
       上下卷扬自动流程:=35;
	35:
	   IF 对中工作完成 THEN
	   	上下卷扬自动流程:=10;
	   END_IF
	40:
	   IF ABS(上侧距离-下侧距离)>50  THEN
	   	   IF 上侧距离>下侧距离 THEN
	   	   	  上下侧距离差值:=上侧距离-下侧距离;
			  上卷扬伺服参数.运行位置:=上卷扬.fActPosition+(上下侧距离差值/10);
			  上卷扬伺服参数.运行模式:=2;
			  上下卷扬自动流程:=50;
		   ELSE
		      上下侧距离差值:=下侧距离-上侧距离;
			  下卷扬伺服参数.运行位置:=下卷扬.fActPosition+(上下侧距离差值/10);
			  下卷扬伺服参数.运行模式:=2;
			  上下卷扬自动流程:=50;
	   	   END_IF
	   ELSE
	       上下卷扬自动流程:=60;
	   END_IF
	50:
	   IF 上卷扬伺服参数.绝对定位状态.DONE OR 下卷扬伺服参数.绝对定位状态.DONE THEN
	   	   上卷扬伺服参数.运行模式:=0;
		   下卷扬伺服参数.运行模式:=0;
		   IF 边沿检测1<>1000 OR 边沿检测2<>1000 OR 边沿检测3<>1000 OR 边沿检测4<>1000 THEN
		   	启动对中机构自动运行:=TRUE;
			上下卷扬自动流程:=55;
		   
           ELSIF ABS(上侧距离-下侧距离)>50  THEN
		   	  上下卷扬自动流程:=40;
		   ELSE
		      上下卷扬自动流程:=80;
		   END_IF
	   END_IF
	55:
	   IF 对中工作完成 THEN
	   	上下卷扬自动流程:=10;
	   END_IF
	60:
	   IF 上侧距离=1000 AND 下侧距离=1000 THEN
	   	   上卷扬伺服参数.运行位置:=20;
		   下卷扬伺服参数.运行位置:=20;
		   上卷扬伺服参数.运行模式:=3;
		   下卷扬伺服参数.运行模式:=3;
		   上下卷扬自动流程:=70;
	   ELSIF 上侧距离=1000  THEN
	       上卷扬伺服参数.运行位置:=20;
		   上卷扬伺服参数.运行模式:=3;
		   上下卷扬自动流程:=70;
	   ELSIF 下侧距离=1000  THEN
	       下卷扬伺服参数.运行位置:=20;
		   下卷扬伺服参数.运行模式:=3;
		   上下卷扬自动流程:=70;
	   ELSE
	       上卷扬伺服参数.运行模式:=0;
		   下卷扬伺服参数.运行模式:=0;
	       上下卷扬自动流程:=80;
	   END_IF
	70:
	   IF 上卷扬伺服参数.相对定位状态.DONE OR 下卷扬伺服参数.相对定位状态.DONE THEN
		   上卷扬伺服参数.运行模式:=0;
		   下卷扬伺服参数.运行模式:=0;
	   	   IF 上侧距离=1000 AND 下侧距离=1000 THEN
			   上下卷扬检测数据有误:=1;
			   上下卷扬自动流程:=1000;
		   ELSIF 边沿检测1<>1000 OR 边沿检测2<>1000 OR 边沿检测3<>1000 OR 边沿检测4<>1000 THEN
		   	启动对中机构自动运行:=TRUE;
			上下卷扬自动流程:=55;
		   ELSE
		       上下卷扬自动流程:=40;
		   END_IF
	   END_IF
	 80:
	   IF 上侧距离>950 OR (上侧距离>上下卷扬距离工作面距离1 AND 上侧距离<950) THEN
			上卷扬伺服参数.运行方向:=TRUE;
			上卷扬伺服参数.运行模式:=1;
			IF 超声波检测左1<上下卷扬距离工作面距离 OR 超声波检测右1<上下卷扬距离工作面距离 THEN
				上卷扬伺服参数.运行模式:=0;
				上卷扬到达清扫面:=TRUE;
			END_IF
	   END_IF
	   IF 下侧距离>950  OR (下侧距离>上下卷扬距离工作面距离1 AND 下侧距离<950) THEN
			下卷扬伺服参数.运行方向:=TRUE;
			下卷扬伺服参数.运行模式:=1;
			IF 超声波检测左2<上下卷扬距离工作面距离 OR 超声波检测右2<上下卷扬距离工作面距离 THEN
				下卷扬伺服参数.运行模式:=0;
				下卷扬到达清扫面:=TRUE;
			END_IF
	   END_IF
	   IF (超声波检测左1<上下卷扬距离工作面距离 OR 超声波检测右1<上下卷扬距离工作面距离) AND (超声波检测左2<上下卷扬距离工作面距离 OR 超声波检测右2<上下卷扬距离工作面距离) THEN
	   	上下卷扬自动流程:=85;
	   END_IF
	 85:
	   	   IF 上侧距离>下侧距离 THEN
	   	   	  上下侧距离差值:=上侧距离-下侧距离;
			  上卷扬伺服参数.运行位置:=上卷扬.fActPosition+(上下侧距离差值/10);
			  上卷扬伺服参数.运行模式:=2;
			  上下卷扬自动流程:=86;
		   ELSE
		      上下侧距离差值:=下侧距离-上侧距离;
			  下卷扬伺服参数.运行位置:=下卷扬.fActPosition+(上下侧距离差值/10);
			  下卷扬伺服参数.运行模式:=2;
			  上下卷扬自动流程:=86;
	   	   END_IF
	 86:
	   IF 上卷扬伺服参数.绝对定位状态.DONE OR 下卷扬伺服参数.绝对定位状态.DONE THEN
	   	   上卷扬伺服参数.运行模式:=0;
		   下卷扬伺服参数.运行模式:=0;
		   上下卷扬自动流程:=88;
	   END_IF
	 87:
	   IF ABS(上侧距离-下侧距离)>5 THEN
	   	上下卷扬自动流程:=88;
	   ELSE
	    上下卷扬自动流程:=90;
	   END_IF
	 88:
	   	   IF 上侧距离>下侧距离 THEN
	   	   	  上下侧距离差值:=上侧距离-下侧距离;
			  上卷扬伺服参数.运行位置:=上卷扬.fActPosition+(上下侧距离差值/10)+补偿值1;
			  上卷扬伺服参数.运行模式:=2;
			  上下卷扬自动流程:=89;
		   ELSE
		      上下侧距离差值:=下侧距离-上侧距离;
			  下卷扬伺服参数.运行位置:=下卷扬.fActPosition+(上下侧距离差值/10)+补偿值2;
			  下卷扬伺服参数.运行模式:=2;
			  上下卷扬自动流程:=89;
	   	   END_IF
	 89:
	   IF 上卷扬伺服参数.绝对定位状态.DONE OR 下卷扬伺服参数.绝对定位状态.DONE THEN
	   
	   	   
		   上下卷扬工作完成:=TRUE;
		   实时检测延时(IN:= TRUE, PT:= 延时时间, Q=> , ET=> );
		   IF 实时检测延时.Q THEN
		       上下卷扬自动流程:=90;
			   实时检测延时(IN:= FALSE, PT:= 延时时间, Q=> , ET=> );
			   上侧距离保存:=上侧距离;
		       下侧距离保存:=下侧距离;
			   上侧实际位置值暂存:=上卷扬.fActPosition;
			   下侧实际位置值暂存:=下卷扬.fActPosition;
		       卷扬1PID复位:=0;
	           卷扬2PID复位:=0;
			   上卷扬伺服参数.运行模式:=0;
		       下卷扬伺服参数.运行模式:=0;
		   END_IF
	   END_IF
	 90://实时监控
	
	        IF 边沿检测1 <> 1000 OR 边沿检测2 <> 1000 THEN
				伸缩轴伺服参数.运行方向:=FALSE;
			    伸缩轴伺服参数.运行模式:=1;
			END_IF
			IF 边沿检测3 <> 1000 OR 边沿检测4 <> 1000 THEN
			    伸缩轴伺服参数.运行方向:=TRUE;
			    伸缩轴伺服参数.运行模式:=1;
			END_IF
	        IF 边沿检测1 = 1000 AND 边沿检测2 = 1000 AND 边沿检测3 = 1000 AND 边沿检测4 = 1000 THEN
		    	伸缩轴伺服参数.运行模式:=0;
		    END_IF
	      
	 
		   上测超声波低通滤波模块(输入数据:= 上侧距离, 滤波系数:= 上下卷扬滤波系数, 输出数据=>上侧滤波距离 );
		   下测超声波低通滤波模块(输入数据:= 下侧距离, 滤波系数:= 上下卷扬滤波系数, 输出数据=>下侧滤波距离 );
		   上测力矩低通滤波模块(输入数据:= adFbForce[1], 滤波系数:= 滤波系数, 输出数据=>上卷扬滤波力矩 );
           下测力矩低通滤波模块(输入数据:= adFbForce[2], 滤波系数:= 滤波系数, 输出数据=>下卷扬滤波力矩 );
		  
		   IF 上侧滤波距离>上下卷扬距离工作面距离1+ 滤波幅值+ 误差限制值 OR 左1滤波距离>600 OR 右1滤波距离>600 THEN
		   	   //上下卷扬自动流程:=100;
			   上卷扬伺服参数.运行位置:=上卷扬.fActPosition ;
		   ELSE
			  // IF 上侧滤波距离>上下卷扬距离工作面距离1+ 滤波幅值 OR 上侧滤波距离<上下卷扬距离工作面距离1- 滤波幅值 THEN
				   (*
				   IF 上侧滤波距离>上下卷扬距离工作面距离1 THEN
					  //上卷扬伺服参数.运行位置:=上卷扬.fActPosition+((上侧滤波距离-上下卷扬距离工作面距离1)/10)*kp设置值;
					  上卷扬伺服参数.运行位置:=上卷扬.fActPosition+(((上侧滤波距离-上下卷扬距离工作面距离1)/10)-上卷扬运行位置保存)*kp设置值+((上侧滤波距离-上下卷扬距离工作面距离1)/10)*ki设置值;
				   ELSE
					  //上卷扬伺服参数.运行位置:=上卷扬.fActPosition-((上下卷扬距离工作面距离1-上侧滤波距离)/10)*kp设置值;
					  上卷扬伺服参数.运行位置:=上卷扬.fActPosition-(((上下卷扬距离工作面距离1-上侧滤波距离)/10)-上卷扬运行位置保存)*kp设置值+((上下卷扬距离工作面距离1-上侧滤波距离)/10)*ki设置值;
				   END_IF
				   上卷扬运行位置保存:=上卷扬伺服参数.运行位置;
				   *)
				   IF 上卷扬滤波力矩 < 上卷扬力矩限制 THEN
			           上卷扬力矩偏差值:=0;
				   ELSE
				       上卷扬力矩偏差值:=-(上卷扬滤波力矩-上卷扬力矩限制);
					   IF 上卷扬力矩偏差值<=-30 THEN
				        	上卷扬力矩偏差值:=-30;
				       END_IF
                   END_IF
				   
				   上卷扬伺服参数.运行位置:=上侧实际位置值暂存+(上侧滤波距离-上下卷扬距离工作面距离1)*ki设置值
				   +(上侧滤波距离-上下卷扬距离工作面距离1-上卷扬运行位置保存)*kp设置值
				   +上卷扬力矩偏差值*力矩kp设置值;
				   上卷扬运行位置保存:=上侧滤波距离-上下卷扬距离工作面距离1;
                   上侧实际位置值暂存:=上卷扬伺服参数.运行位置;
				   //IF (上卷扬.fActPosition>上卷扬上限位 OR 上卷扬.fActPosition<上卷扬下限位) THEN
					   //上卷扬伺服参数.运行位置:=上卷扬.fActPosition ;
				   //END_IF
			 //  END_IF
		   END_IF
		   IF 下侧滤波距离>上下卷扬距离工作面距离1+ 滤波幅值+ 误差限制值 OR 左2滤波距离>600 OR 右2滤波距离>600 THEN
		   	   //上下卷扬自动流程:=100;
			   下卷扬伺服参数.运行位置:=下卷扬.fActPosition;
		   ELSE
			  // IF 下侧滤波距离>上下卷扬距离工作面距离1+ 滤波幅值 OR 下侧滤波距离<上下卷扬距离工作面距离1- 滤波幅值 THEN
				   (*
				   IF 下侧滤波距离>上下卷扬距离工作面距离1 THEN
					  //下卷扬伺服参数.运行位置:=下卷扬.fActPosition+((下侧滤波距离-上下卷扬距离工作面距离1)/10)*kp设置值;
					  下卷扬伺服参数.运行位置:=下卷扬.fActPosition+(((下侧滤波距离-上下卷扬距离工作面距离1)/10)-下卷扬运行位置保存)*kp设置值+((下侧滤波距离-上下卷扬距离工作面距离1)/10)*ki设置值;
				   ELSE
					  //下卷扬伺服参数.运行位置:=下卷扬.fActPosition-((上下卷扬距离工作面距离1-下侧滤波距离)/10)*kp设置值;
					  下卷扬伺服参数.运行位置:=下卷扬.fActPosition-(((上下卷扬距离工作面距离1-下侧滤波距离)/10)-下卷扬运行位置保存)*kp设置值+((上下卷扬距离工作面距离1-下侧滤波距离)/10)*ki设置值;
				   END_IF
				   下卷扬运行位置保存:=下卷扬伺服参数.运行位置;
				   *)
				   IF 下卷扬滤波力矩 < 下卷扬力矩限制 THEN
			           下卷扬力矩偏差值:=0;
				   ELSE
				       下卷扬力矩偏差值:=-(下卷扬滤波力矩-下卷扬力矩限制);
					   IF 下卷扬力矩偏差值<=-30 THEN
				        	下卷扬力矩偏差值:=-30;
				       END_IF
                   END_IF
				   下卷扬伺服参数.运行位置:=下侧实际位置值暂存+(下侧滤波距离-上下卷扬距离工作面距离1)*ki设置值
				   +(下侧滤波距离-上下卷扬距离工作面距离1-下卷扬运行位置保存)*kp设置值
				   +下卷扬力矩偏差值*力矩kp设置值1;
				   下卷扬运行位置保存:=下侧滤波距离-上下卷扬距离工作面距离1;
                   下侧实际位置值暂存:=下卷扬伺服参数.运行位置;
				  // IF (下卷扬.fActPosition>下卷扬上限位 OR 下卷扬.fActPosition<下卷扬下限位) THEN
					   //下卷扬伺服参数.运行位置:=下卷扬.fActPosition;
				   //END_IF
			  // END_IF
		   END_IF
	       上卷扬实时控制(超声波实时检测:= TRUE, 运行位置:= 上卷扬伺服参数.运行位置, 伺服参数:= 上卷扬伺服参数);
	       下卷扬实时控制(超声波实时检测:= TRUE, 运行位置:= 下卷扬伺服参数.运行位置, 伺服参数:= 下卷扬伺服参数);
		   //上下卷扬工作完成:=TRUE;
		   (*
	       IF (超声波检测左1=1000 AND 超声波检测左2=1000) OR (超声波检测右1=1000 AND 超声波检测右2=1000) 
			   OR 超声波检测左1>上下卷扬距离工作面距离1+70 OR 超声波检测左2>上下卷扬距离工作面距离1+70
			   OR 超声波检测右1>上下卷扬距离工作面距离1+70 OR 超声波检测右2>上下卷扬距离工作面距离1+70 THEN
				   
	       	;
	       END_IF
	       *)
	(* 
	 90:
	   上下卷扬工作完成:=TRUE;
	   上卷扬伺服参数.运行模式:=0;
	   下卷扬伺服参数.运行模式:=0;
	   启动上下扬自动运行:=FALSE;
	   上下卷扬自动流程:=0;
	  *) 
	  100:
	      上卷扬伺服参数.运行模式:=10;
		  下卷扬伺服参数.运行模式:=10;
		  伸缩轴伺服参数.运行模式:=10;
		  上下卷扬工作完成:=FALSE;
		  上下卷扬异常:=TRUE;
	 
	  110:
	      IF 上侧距离 <> 1000  THEN		
		     卷扬1处理数值 := LREAL_TO_REAL (上侧距离);	
	      ELSE
		     卷扬1处理数值 := LREAL_TO_REAL (上侧距离保存);
	      END_IF
		  IF 下侧距离 <> 1000  THEN
		     卷扬2处理数值 := LREAL_TO_REAL (下侧距离);
	      ELSE
		     卷扬2处理数值 := LREAL_TO_REAL (下侧距离保存);
	      END_IF
		  
		  IF  ABS(上侧距离保存 - 卷扬1处理数值) <= 卷扬1PID.允许偏差 THEN
			    上卷扬伺服参数.运行模式:=5;
				上卷扬速度控制(启动底盘自动运行:= FALSE, 伺服参数:= 上卷扬伺服参数); 
			 	卷扬1到位 :=1;				
		  ELSE
			    卷扬1到位 :=0;
				上卷扬速度控制(启动底盘自动运行:= TRUE, 伺服参数:= 上卷扬伺服参数); 
			    上卷扬伺服参数.运行速度 := PID_1.Y;	
				IF 上卷扬伺服参数.运行速度>0 THEN
					上卷扬伺服参数.运行控制方向:=1;
				ELSIF 上卷扬伺服参数.运行速度<0 THEN
				    上卷扬伺服参数.运行控制方向:=-1;
				ELSE
				    上卷扬伺服参数.运行模式:=5;
				END_IF
		  END_IF		
		
		  IF 卷扬1到位 THEN
			   卷扬1处理数值 := 上侧距离保存;
		  END_IF
		  
		  
		  IF  ABS(下侧距离保存 - 卷扬2处理数值) <= 卷扬2PID.允许偏差 THEN
			    下卷扬伺服参数.运行模式:=5;
				下卷扬速度控制(启动底盘自动运行:= FALSE, 伺服参数:= 下卷扬伺服参数); 
			 	卷扬2到位 :=1;				
		  ELSE
			    卷扬2到位 :=0;
				下卷扬速度控制(启动底盘自动运行:= TRUE, 伺服参数:= 下卷扬伺服参数); 
			    下卷扬伺服参数.运行速度 := PID_2.Y;	
				IF 下卷扬伺服参数.运行速度>0 THEN
					下卷扬伺服参数.运行控制方向:=1;
				ELSIF 下卷扬伺服参数.运行速度<0 THEN
				    下卷扬伺服参数.运行控制方向:=-1;
				ELSE
				    下卷扬伺服参数.运行模式:=5;
				END_IF
		  END_IF		
		
		  IF 卷扬2到位 THEN
			   卷扬2处理数值 := 下侧距离保存;
		  END_IF
		
		  
	 1000:
	   ;
ELSE
	;
END_CASE

       PID_1(
				ACTUAL:= LREAL_TO_REAL(卷扬1处理数值), 
				SET_POINT:= LREAL_TO_REAL(上侧距离保存), 
				KP:= 卷扬1PID.KP, 
				TN:= 卷扬1PID.TN, 
				TV:= 卷扬1PID.TV, 
				Y_MANUAL:= , 
				Y_OFFSET:= , 
				Y_MIN:= 卷扬1PID.输出最小值, 
				Y_MAX:= 卷扬1PID.输出最大值,
				MANUAL:= , 
				RESET:= 卷扬1PID复位, 
				Y=> , 
				LIMITS_ACTIVE=> , 
				OVERFLOW=> );	
				
		  PID_2(
				ACTUAL:= LREAL_TO_REAL(卷扬2处理数值), 
				SET_POINT:= LREAL_TO_REAL(下侧距离保存), 
				KP:= 卷扬2PID.KP, 
				TN:= 卷扬2PID.TN, 
				TV:= 卷扬2PID.TV, 
				Y_MANUAL:= , 
				Y_OFFSET:= , 
				Y_MIN:= 卷扬2PID.输出最小值, 
				Y_MAX:= 卷扬2PID.输出最大值, 
				MANUAL:= , 
				RESET:= 卷扬2PID复位, 
				Y=> , 
				LIMITS_ACTIVE=> , 
				OVERFLOW=> );	
				
ELSE
      上下卷扬检测数据有误:=FALSE;
	   上卷扬到达清扫面:=FALSE;
	   下卷扬到达清扫面:=FALSE;
	   上下卷扬工作完成:=FALSE;
	   上下卷扬自动流程:=0;
	   //上卷扬伺服参数.运行模式:=0;
	   //下卷扬伺服参数.运行模式:=0;
	   上卷扬实时控制(超声波实时检测:= FALSE, 运行位置:= 上卷扬伺服参数.运行位置, 伺服参数:= 上卷扬伺服参数);
	   下卷扬实时控制(超声波实时检测:= FALSE, 运行位置:= 下卷扬伺服参数.运行位置, 伺服参数:= 下卷扬伺服参数);
	 
END_IF
END_ACTION

ACTION 传感器检测:
//假如8个传感器都没有值另外处理
{region}//模拟量
//检测传感器数值，转换为距离

IF (i_模拟量1 <=19600) AND (i_模拟量1 >= 0)  THEN
	//边沿检测1 
	边沿检测1 := (INT_TO_REAL(i_模拟量1) / 19692) * (1000 -60) +60;
ELSE
	边沿检测1 := 1000;
END_IF

IF (i_模拟量2 <=19600) AND (i_模拟量2 >= 0) THEN
	//边沿检测2
	边沿检测2 := (INT_TO_REAL(i_模拟量2) / 19692) * (1000 -60) +60;
ELSE
	边沿检测2 := 1000;
END_IF

IF (i_模拟量7 <=19600) AND (i_模拟量7 >= 0)  THEN
	//边沿检测3
	边沿检测3 := (INT_TO_REAL(i_模拟量7) / 19692) * (1000 -60) +60;
ELSE
	边沿检测3 := 1000;
END_IF

IF (i_模拟量8 <=19600) AND (i_模拟量8 >= 0) THEN
	//边沿检测4
	边沿检测4 := (INT_TO_REAL(i_模拟量8) / 19692) * (1000 -60) +60;
ELSE
	边沿检测4 := 1000;
END_IF

IF (i_模拟量3 <=19600) AND (i_模拟量3 >=0) THEN
	//超声波检测左1
	超声波检测左1 := (INT_TO_REAL(i_模拟量3) / 19692) * (1000 -60) +60;
ELSE
	超声波检测左1 := 1000;
END_IF

IF (i_模拟量4 <=19600) AND  (i_模拟量4 >=0) THEN
	//超声波检测左2
	超声波检测右1 := (INT_TO_REAL(i_模拟量4) / 19692) * (1000 -60) +60;
ELSE
	超声波检测右1 := 1000;
END_IF

IF (i_模拟量5 <=19600) AND  (i_模拟量5 >=0) THEN
	//超声波检测右1
	超声波检测左2 := (INT_TO_REAL(i_模拟量5) / 19692) * (1000 -60) +60;
ELSE
	超声波检测左2 := 1000;
END_IF

IF (i_模拟量6 <=19600) AND  (i_模拟量6 >=0) THEN
	//超声波检测右2
	超声波检测右2 := (INT_TO_REAL(i_模拟量6) / 19692) * (1000 -60) +60;
ELSE
	超声波检测右2 := 1000;
END_IF

左1超声波低通滤波模块(输入数据:= 超声波检测左1, 滤波系数:= 上下卷扬滤波系数, 输出数据=>左1滤波距离 );
左2超声波低通滤波模块(输入数据:= 超声波检测左2, 滤波系数:= 上下卷扬滤波系数, 输出数据=>左2滤波距离 );
右1超声波低通滤波模块(输入数据:= 超声波检测右1, 滤波系数:= 上下卷扬滤波系数, 输出数据=>右1滤波距离 );
右2超声波低通滤波模块(输入数据:= 超声波检测右2, 滤波系数:= 上下卷扬滤波系数, 输出数据=>右2滤波距离 );

//上侧距离测量，有一侧或者两侧都没在范围内
IF 左1滤波距离 = 1000 OR 右1滤波距离 =1000 THEN//检测不到默认值为1000
	IF 左1滤波距离 = 1000 THEN
		上侧距离 := 右1滤波距离;
	ELSE
		上侧距离 := 左1滤波距离;	
	END_IF
ELSE//两个传感器都检测到有距离值，两侧都在范围内，但是大于超声波允许相差长度
	IF ABS(左1滤波距离 - 右1滤波距离) > 50 THEN
		IF 左1滤波距离 < 右1滤波距离 THEN
			上侧距离 := 左1滤波距离;
		ELSE
			上侧距离 := 右1滤波距离;
		END_IF
	ELSE
		上侧距离 := (左1滤波距离 + 右1滤波距离) / 2;
	END_IF
	
END_IF

//下侧距离测量，有一侧或者两侧都没在范围内
IF 右2滤波距离 = 1000 OR 左2滤波距离 =1000 THEN
	IF 超声波检测右2 = 1000 THEN
		下侧距离 := 左2滤波距离;
	ELSE
		下侧距离 := 右2滤波距离;	
	END_IF
ELSE//两个传感器都检测到有距离值，两侧都在范围内，但是大于超声波允许相差长度
	IF ABS(左2滤波距离 - 右2滤波距离) > 50 THEN
		IF 左2滤波距离 < 右2滤波距离 THEN
			下侧距离 := 左2滤波距离;
		ELSE
			下侧距离 := 右2滤波距离;
		END_IF
	ELSE
		下侧距离 := (右2滤波距离 + 左2滤波距离) / 2;
	END_IF
END_IF

IF 超声波检测左1=1000 OR 超声波检测右1=1000 OR 超声波检测左2=1000 OR 超声波检测右2=1000 THEN
	   	IF 超声波检测左1<>1000 AND 超声波检测左2<>1000 AND 超声波检测右1=1000 AND 超声波检测右2=1000 THEN
	   		上侧距离:=超声波检测左1;
			下侧距离:=超声波检测左2;
		ELSIF 超声波检测右1<>1000 AND 超声波检测右2<>1000 AND 超声波检测左1=1000 AND 超声波检测左2=1000 THEN
	   		上侧距离:=超声波检测右1;
			下侧距离:=超声波检测右2;
		ELSIF 超声波检测左1<>1000 AND 超声波检测左2<>1000 AND 超声波检测右1<>1000 AND 超声波检测右2=1000 THEN
	   		上侧距离:=超声波检测左1;
			下侧距离:=超声波检测左2;
		ELSIF 超声波检测左1<>1000 AND 超声波检测左2<>1000 AND 超声波检测右1=1000 AND 超声波检测右2<>1000 THEN
	   		上侧距离:=超声波检测左1;
			下侧距离:=超声波检测左2;
		ELSIF 超声波检测右1<>1000 AND 超声波检测右2<>1000 AND 超声波检测左1<>1000 AND 超声波检测左2=1000 THEN
	   		上侧距离:=超声波检测右1;
			下侧距离:=超声波检测右2;
		ELSIF 超声波检测右1<>1000 AND 超声波检测右2<>1000 AND 超声波检测左1=1000 AND 超声波检测左2<>1000 THEN
	   		上侧距离:=超声波检测右1;
			下侧距离:=超声波检测右2;
	   	END_IF;
	   END_IF
END_ACTION

ACTION 对中机构控制:
//对中机构
IF 启动对中机构自动运行 THEN
	CASE 对中机构自动流程 OF
		0:
		    对中工作完成 :=FALSE;
			伸缩轴伺服参数.运行模式:=0;
			伸缩轴伺服参数.运行速度:=10;
			对中机构自动流程:=10;
		10:
			IF 边沿检测1 = 1000 AND 边沿检测2 = 1000 AND 边沿检测3 = 1000 AND 边沿检测4 = 1000 THEN
				对中工作完成 :=TRUE;
				对中机构自动流程:=70;
			ELSE
				对中机构自动流程:=20;
			END_IF;
		20:	
		    IF 边沿检测1 <> 1000 OR 边沿检测2 <> 1000 THEN
				伸缩轴伺服参数.运行方向:=FALSE;
			    伸缩轴伺服参数.运行模式:=1;
				对中机构自动流程:=30;
			END_IF
			IF 边沿检测3 <> 1000 OR 边沿检测4 <> 1000 THEN
			    伸缩轴伺服参数.运行方向:=TRUE;
			    伸缩轴伺服参数.运行模式:=1;
				对中机构自动流程:=50;
			END_IF
		30:
		    IF 边沿检测1 = 1000 AND 边沿检测2 = 1000 THEN
		    	伸缩轴伺服参数.运行模式:=0;
				对中机构自动流程:=40;
		    END_IF
		40:
		    伸缩轴伺服参数.运行位置:=伸缩轴.fActPosition-50;
		    伸缩轴伺服参数.运行模式:=2;
			对中机构自动流程:=45;
		45:
			IF 伸缩轴伺服参数.绝对定位状态.DONE THEN
				伸缩轴伺服参数.运行模式:=0;
				对中机构自动流程:=0;
			END_IF
		50:
		    IF 边沿检测3 = 1000 AND 边沿检测4 = 1000 THEN
		    	伸缩轴伺服参数.运行模式:=0;
				对中机构自动流程:=60;
		    END_IF
		60:
		    伸缩轴伺服参数.运行位置:=伸缩轴.fActPosition+50;
		    伸缩轴伺服参数.运行模式:=2;
			对中机构自动流程:=65;
		65:
			IF 伸缩轴伺服参数.绝对定位状态.DONE THEN
				伸缩轴伺服参数.运行模式:=0;
				对中机构自动流程:=0;
			END_IF
		70:
		    对中工作完成:=TRUE;
			启动对中机构自动运行:=FALSE;
			对中机构自动流程:=0;
	 END_CASE	
ELSE
            对中工作完成 :=FALSE;
			//伸缩轴伺服参数.运行模式:=0;
			伸缩轴伺服参数.运行速度:=10;
			对中机构自动流程:=0;
END_IF
END_ACTION

ACTION 回零控制:
IF 启动回零自动运行 THEN
	CASE 回零自动流程 OF
		0:
		   回零工作完成:=FALSE;
		   上卷扬回零完成:=FALSE;
		   下卷扬回零完成:=FALSE;
		   伸缩架回零完成:=FALSE;
		   上卷扬零点位置:=-1251.0;
	       下卷扬零点位置:=-2545.0;
	       伸缩架零点位置:=30.0;
		   回零自动流程:=10;
		   上卷扬伺服参数.运行模式:=0;
		   下卷扬伺服参数.运行模式:=0;
		   伸缩轴伺服参数.运行模式:=0;
		   上卷扬伺服参数.绝对定位状态.DONE:=FALSE;
		   下卷扬伺服参数.绝对定位状态.DONE:=FALSE;
		   伸缩轴伺服参数.绝对定位状态.DONE:=FALSE;
		10:
		   IF 回零工作完成=FALSE THEN
			   上卷扬伺服参数.运行位置:=上卷扬零点位置;
			   下卷扬伺服参数.运行位置:=下卷扬零点位置;
			   伸缩轴伺服参数.运行位置:=伸缩架零点位置;
			   滚刷伺服参数.运行模式:=0;
			   上卷扬伺服参数.运行模式:=2;
			   下卷扬伺服参数.运行模式:=2;
			   伸缩轴伺服参数.运行模式:=2;
			   回零自动流程:=20;
		   END_IF
		 20:
		   IF 上卷扬伺服参数.绝对定位状态.DONE THEN
		   	   上卷扬回零完成:=TRUE;
		   END_IF
		   IF 下卷扬伺服参数.绝对定位状态.DONE THEN
		   	   下卷扬回零完成:=TRUE;
		   END_IF
		   IF 伸缩轴伺服参数.绝对定位状态.DONE THEN
		   	   伸缩架回零完成:=TRUE;
		   END_IF
		   IF 上卷扬回零完成 AND 下卷扬回零完成 AND 伸缩架回零完成 THEN
			   回零工作完成:=TRUE;
		   	   回零自动流程:=30;
		   END_IF
		 30:
		   启动回零自动运行:=FALSE;
		   回零自动流程:=0;
	END_CASE
ELSE
           回零工作完成:=FALSE;
		   上卷扬回零完成:=FALSE;
		   下卷扬回零完成:=FALSE;
		   伸缩架回零完成:=FALSE;
		   上卷扬零点位置:=-30;
	       下卷扬零点位置:=-50;
	       伸缩架零点位置:=-30;
		   回零自动流程:=0;
END_IF
END_ACTION

ACTION 报警检测:
//报警触发
//限位触发
END_ACTION

ACTION 滚刷控制:
IF 启动滚刷自动运行 THEN
	IF 滚刷正转 THEN
		滚刷伺服参数.运行方向:=TRUE;
		滚刷伺服参数.运行模式:=1;
	END_IF;
	IF 滚刷反转 THEN
		滚刷伺服参数.运行方向:=FALSE;
		滚刷伺服参数.运行模式:=1;
	END_IF;
ELSE
    滚刷伺服参数.运行模式:=0;
END_IF
END_ACTION

ACTION ACT_test:
CASE 上下卷扬自动流程 OF
	0:
		上侧实际位置值暂存:=100;
		下侧实际位置值暂存:=100;
		//上下卷扬自动流程:=10;
	10:
	    上卷扬伺服参数.运行位置:=上侧实际位置值暂存+(上侧滤波距离-上下卷扬距离工作面距离1)*kp设置值+(上侧滤波距离-上下卷扬距离工作面距离1-上卷扬运行位置保存)*ki设置值;
		上卷扬运行位置保存:=上侧滤波距离-上下卷扬距离工作面距离1;
        上侧实际位置值暂存:=上卷扬伺服参数.运行位置;
END_CASE
END_ACTION

END_PROGRAM

// Device/Application/电池数据通讯
PROGRAM 电池数据通讯
VAR
	iCounter : INT := 0;
END_VAR

系统状态 := WORD_TO_INT(BMS映射数据[0]); // 0-初始化 1-待机模式 2-充电模式 3-放电模式 4-上电BCU编码中 5-上电BMU编码中 6-上电绝缘检测中 7-上电并机中 8-掉电中 9-系统锁定
电池状态 := WORD_TO_INT(BMS映射数据[1]); // 0-等待 1-禁充禁放 2-禁充 3-禁放 4-充电中 5-放电中
一级保护状态 := SHL(BMS映射数据[2], 16) OR BMS映射数据[3];
二级保护状态 := SHL(BMS映射数据[4], 16) OR BMS映射数据[5];
三级保护状态 := SHL(BMS映射数据[6], 16) OR BMS映射数据[7];
故障状态 := SHL(BMS映射数据[8], 16) OR BMS映射数据[9];
采集电压 := WORD_TO_LREAL(BMS映射数据[10]) * 0.1; 		// 转换为V
负载电压 := WORD_TO_LREAL(BMS映射数据[11]) * 0.1; 		// 转换为V
上桥累计电压 := WORD_TO_LREAL(BMS映射数据[12]) * 0.1; 	// 转换为V
下桥累计电压 := WORD_TO_LREAL(BMS映射数据[13]) * 0.1; 	// 转换为V
上桥电流 := DWORD_TO_DINT(SHL(BMS映射数据[14], 16) OR BMS映射数据[15]) * 0.01; // 转换为A
下桥电流 := DWORD_TO_DINT(SHL(BMS映射数据[16], 16) OR BMS映射数据[17]) * 0.01; // 转换为A
上桥SOC := WORD_TO_LREAL(BMS映射数据[18]); // 单位%
下桥SOC := WORD_TO_LREAL(BMS映射数据[19]); // 单位%
上桥SOH := WORD_TO_LREAL(BMS映射数据[20]); // 单位%
下桥SOH := WORD_TO_LREAL(BMS映射数据[21]); // 单位%
上桥电池剩余容量 := DWORD_TO_DINT(SHL(BMS映射数据[22], 16) OR BMS映射数据[23]) * 0.01; // 单位AH
下桥电池剩余容量 := DWORD_TO_DINT(SHL(BMS映射数据[24], 16) OR BMS映射数据[25]) * 0.01; // 单位AH
上桥系统功率 := WORD_TO_LREAL(BMS映射数据[26]) * 0.1; // 单位KW
下桥系统功率 := WORD_TO_LREAL(BMS映射数据[27]) * 0.1; // 单位KW

UPS警告项1 := UPS映射数据[0];
UPS警告项2 := UPS映射数据[1];
UPS警告项3 := UPS映射数据[2];
UPS警告项4 := UPS映射数据[3];
UPS警告项5 := UPS映射数据[4];
R输入电压 := WORD_TO_LREAL(UPS映射数据[5]) * 0.01804; 		// 转换为V
S输入电压 := WORD_TO_LREAL(UPS映射数据[6]) * 0.01804; 		// 转换为V
T输入电压 := WORD_TO_LREAL(UPS映射数据[7]) * 0.01804; 		// 转换为V
R输出电压 := WORD_TO_LREAL(UPS映射数据[9]) * 0.1; 			// 转换为V
S输出电压 := WORD_TO_LREAL(UPS映射数据[10]) * 0.1; 		// 转换为V
T输出电压 := WORD_TO_LREAL(UPS映射数据[11]) * 0.1; 		// 转换为V
输出频率 := WORD_TO_LREAL(UPS映射数据[12]) * 0.1; 			// 转换为Hz
R输出电流 := WORD_TO_LREAL(UPS映射数据[13]) * 0.1; 		// 转换为A
S输出电流 := WORD_TO_LREAL(UPS映射数据[14]) * 0.1; 		// 转换为A
T输出电流 := WORD_TO_LREAL(UPS映射数据[15]) * 0.1; 		// 转换为A
R输出负载百分比 := WORD_TO_LREAL(UPS映射数据[16]) * 0.1; 	// 转换为%
S输出负载百分比 := WORD_TO_LREAL(UPS映射数据[17]) * 0.1; 	// 转换为%
T输出负载百分比 := WORD_TO_LREAL(UPS映射数据[18]) * 0.1; 	// 转换为%
总输出负载百分比 := WORD_TO_LREAL(UPS映射数据[19]) * 0.1; 	// 转换为%
UPS状态 := UPS映射数据[20];
散热器温度1 := WORD_TO_LREAL(UPS映射数据[21]); // 转换为度
散热器温度2 := WORD_TO_LREAL(UPS映射数据[22]); // 转换为度
机柜温度 := WORD_TO_LREAL(UPS映射数据[23]); 	// 转换为度
UPS模式 := UPS映射数据[24]; //0x50-开机模式 0x53-待机模式 0x59-旁路模式 0x4C-线路模式 0x42-电池模式 0x46-故障模式 0x45-HE/ECO模式 0x43-转换器模式 0x44-关机模式 
UPS故障信息 := UPS映射数据[25];
当前功率 := WORD_TO_LREAL(UPS映射数据[26]); 	// 转换为W

FOR iCounter:=0 TO 29 BY 1 DO
	电池反馈电压组1[iCounter] := WORD_TO_LREAL(电池映射电压组1[iCounter]) * 0.001; // 转换为V
	电池反馈电压组2[iCounter] := WORD_TO_LREAL(电池映射电压组2[iCounter]) * 0.001; // 转换为V
	电池反馈电压组3[iCounter] := WORD_TO_LREAL(电池映射电压组3[iCounter]) * 0.001; // 转换为V
	电池反馈电压组4[iCounter] := WORD_TO_LREAL(电池映射电压组4[iCounter]) * 0.001; // 转换为V
END_FOR

FOR iCounter:=0 TO 9 BY 1 DO
	电池反馈温度组1[iCounter] := 电池映射温度组1[iCounter] * 0.1; // 转换为度
	电池反馈温度组2[iCounter] := 电池映射温度组2[iCounter] * 0.1; // 转换为度
	电池反馈温度组3[iCounter] := 电池映射温度组3[iCounter] * 0.1; // 转换为度
	电池反馈温度组4[iCounter] := 电池映射温度组4[iCounter] * 0.1; // 转换为度
END_FOR

IF 上桥SOC<15 OR 下桥SOC<15 THEN
	电量报警 := TRUE;
// 	电量状态 := 0;
ELSIF 上桥SOC>95 OR 下桥SOC>95 THEN
	电量报警 := FALSE;
// 	电量状态 := 2;
ELSE
	电量报警 := FALSE;
// 	电量状态 := 1;
END_IF

END_PROGRAM

// Device/Application/DCH遥控控制
PROGRAM DCH遥控控制
VAR
	//DCH读数据
	DCH无线状态		: BOOL;
	DCH急停			: BOOL;
	DCH遥控			: BOOL;
	DCH本地			: BOOL;
	DMI控制			: BOOL;
	DCH电机控制0 		: BOOL;
	DCH电机控制1 		: BOOL;
	DCH电机控制2 		: BOOL;
	DCH电机控制3 		: BOOL;
	DCH滚刷正转		: BOOL;
	DCH滚刷关闭		: BOOL;
	DCH滚刷反转		: BOOL;
	DCH启动			: BOOL;
	DCH停止			: BOOL;
	DCH伺服ON		: BOOL;
	DCH伺服OFF		: BOOL;
	DCH_F1			: BOOL;
	DCH_F2			: BOOL;
	
	DCH前进			: BOOL;
	DCH后退			: BOOL;
	DCH左转			: BOOL;
	DCH右转			: BOOL;
	DCH方向1正转		: BOOL;
	DCH方向1反转		: BOOL;
	DCH方向2正转		: BOOL;
	DCH方向2反转		: BOOL;
	DCH方向3正转		: BOOL;
	DCH方向3反转		: BOOL;
	DCH方向4正转		: BOOL;
	DCH方向4反转		: BOOL;
	
	DCH前后数值量		: LREAL;
	DCH左右数值量		: LREAL;
	DCH方向1数值量	: LREAL;
	DCH方向2数值量	: LREAL;
	DCH方向3数值量	: LREAL;
	DCH方向4数值量	: LREAL;
	
	//DCH写数据
	DCH状态位		: WORD;	
	DCH状态位_自动	: BOOL;
	DCH状态位_手动	: BOOL;
	DCH状态位_运行	: BOOL;
	DCH状态位_报警	: BOOL;
	DCH状态位_急停	: BOOL;
	DCH状态位_边沿1	: BOOL;
	DCH状态位_边沿2	: BOOL;
	
	DCH上测距		: INT;
	DCH下测距		: INT;
	
	发动机启动定时器      : TON;
	发动机开关定时器      : TON;
	发动机启动定时器开关   : BOOL := FALSE;
	发动机开关定时器开关   : BOOL := FALSE;
	发动机开关		: BOOL := FALSE;
	发动机启动		: BOOL := FALSE;
	机械臂手动运行	: BOOL := FALSE;
END_VAR

DCH遥控数值刷新();

IF DCH无线状态=FALSE THEN
	RETURN;
END_IF

IF DCH急停=TRUE THEN
	机械臂使能 := FALSE;
	底盘使能 := FALSE;
	末端使能 := FALSE;
	DCH状态位_急停 := TRUE;
ELSE
	DCH状态位_急停 := FALSE;
END_IF

IF DCH_F1=TRUE THEN
	报警复位 := TRUE;
ELSE
	报警复位 := FALSE;
END_IF

IF DCH_F2=TRUE OR (报警代码4.0 AND 报警代码4.1 )THEN
	发动机开关定时器开关 := TRUE;
	发动机启动定时器开关 := TRUE;
END_IF

IF 发动机开关定时器.Q THEN
	发动机开关 := NOT(发动机开关);
	发动机开关定时器开关 := FALSE;
END_IF

IF 发动机启动定时器.Q THEN
	发动机启动 := NOT(发动机启动);
	发动机启动定时器开关 := FALSE;
END_IF
发动机开关定时器(IN:= 发动机开关定时器开关, PT:= T#5S, Q=> , ET=> );
发动机启动定时器(IN:= 发动机启动定时器开关, PT:= T#12S, Q=> , ET=> );

IF DCH遥控=TRUE THEN
	控制方式 := 1;	//自动模式
ELSE
	控制方式 := 0;	//手动模式
END_IF

IF DCH本地=FALSE THEN
	DCH状态位_手动 := FALSE;
	DCH状态位_自动 := TRUE;
	RETURN;
END_IF

DCH状态位_手动 := TRUE;
DCH状态位_自动 := FALSE;

IF DCH伺服ON=TRUE THEN
	机械臂使能 := TRUE;
	底盘使能 := TRUE;
	末端使能 := TRUE;
	DCH状态位_运行 := TRUE;
END_IF

IF DCH伺服OFF=TRUE THEN
	机械臂使能 := FALSE;
	底盘使能 := FALSE;
	末端使能 := FALSE;
	DCH状态位_运行 := FALSE;
END_IF

DCH底盘控制();
DCH机械臂控制();
DCH末端控制();

METHOD DCH末端控制
VAR_INPUT
END_VAR
IF DCH电机控制3=FALSE THEN
	RETURN;
END_IF

IF DCH启动=TRUE THEN
	启动回零自动运行 := TRUE;
END_IF

IF 启动回零自动运行=TRUE THEN
	RETURN;
END_IF

IF DCH方向1正转 OR DCH方向1反转 THEN
	IF DCH方向1正转=TRUE THEN
		伸缩轴伺服参数.运行模式 := 1;
		伸缩轴伺服参数.运行方向 := FALSE;
	END_IF
	IF DCH方向1反转=TRUE THEN
		伸缩轴伺服参数.运行模式 := 1;
		伸缩轴伺服参数.运行方向 := TRUE;
	END_IF
ELSE
	伸缩轴伺服参数.运行模式 := 0;
END_IF

IF DCH方向2正转 OR DCH方向2反转 THEN
	IF DCH方向2正转=TRUE THEN
		上卷扬伺服参数.运行模式 := 1;
		上卷扬伺服参数.运行方向 := TRUE;
	END_IF
	IF DCH方向2反转=TRUE THEN
		上卷扬伺服参数.运行模式 := 1;
		上卷扬伺服参数.运行方向 := FALSE;
	END_IF
ELSE
	上卷扬伺服参数.运行模式 := 0;
END_IF

IF DCH方向3正转 OR DCH方向3反转 THEN
	IF DCH方向3正转=TRUE THEN
		下卷扬伺服参数.运行模式 := 1;
		下卷扬伺服参数.运行方向 := TRUE;
	END_IF
	IF DCH方向3反转=TRUE THEN
		下卷扬伺服参数.运行模式 := 1;
		下卷扬伺服参数.运行方向 := FALSE;
	END_IF
ELSE
	下卷扬伺服参数.运行模式 := 0;
END_IF

IF DCH方向4正转 OR DCH方向4反转 THEN
	IF DCH方向4正转=TRUE THEN
		滚刷伺服参数.运行模式 := 1;
		滚刷伺服参数.运行方向 := TRUE;
	END_IF
	IF DCH方向4反转=TRUE THEN
		滚刷伺服参数.运行模式 := 1;
		滚刷伺服参数.运行方向 := FALSE;
	END_IF
ELSE
	滚刷伺服参数.运行模式 := 0;
END_IF
END_METHOD

METHOD DCH遥控数值刷新
VAR_INPUT
END_VAR
DCH无线状态 := DCH读遥控数据[6].1;
DCH急停 := NOT(DCH读遥控数据[7].12);
DCH遥控 := DCH读遥控数据[6].15;
DCH本地 := DCH读遥控数据[6].14;
DMI控制 := NOT(DCH读遥控数据[6].14 OR DCH读遥控数据[6].15);
DCH电机控制0 := DCH读遥控数据[7].0;
DCH电机控制1 := DCH读遥控数据[7].1;
DCH电机控制2 := DCH读遥控数据[7].2;
DCH电机控制3 := DCH读遥控数据[7].3;
DCH滚刷正转 := DCH读遥控数据[7].4;
DCH滚刷反转 := DCH读遥控数据[7].5;
DCH滚刷关闭 := NOT(DCH读遥控数据[7].4 OR DCH读遥控数据[7].5);
DCH启动 := DCH读遥控数据[7].6;
DCH停止 := DCH读遥控数据[7].7;
DCH伺服ON := DCH读遥控数据[7].9;
DCH伺服OFF := DCH读遥控数据[7].10;
DCH_F1 := DCH读遥控数据[7].8;
DCH_F2 := DCH读遥控数据[7].11;
DCH前进 := DCH读遥控数据[6].2;
DCH后退 := DCH读遥控数据[6].3;
DCH左转 := DCH读遥控数据[6].5;
DCH右转 := DCH读遥控数据[6].4;
DCH方向1正转 := DCH读遥控数据[6].6;
DCH方向1反转 := DCH读遥控数据[6].7;
DCH方向2正转 := DCH读遥控数据[6].8;
DCH方向2反转 := DCH读遥控数据[6].9;
DCH方向3正转 := DCH读遥控数据[6].10;
DCH方向3反转 := DCH读遥控数据[6].11;
DCH方向4正转 := DCH读遥控数据[6].12;
DCH方向4反转 := DCH读遥控数据[6].13;

DCH前后数值量 := WORD_TO_LREAL(DCH读遥控数据[0]);
DCH左右数值量 := WORD_TO_LREAL(DCH读遥控数据[1]);
DCH方向1数值量 := WORD_TO_LREAL(DCH读遥控数据[2]);
DCH方向2数值量 := WORD_TO_LREAL(DCH读遥控数据[3]);
DCH方向3数值量 := WORD_TO_LREAL(DCH读遥控数据[4]);
DCH方向4数值量 := WORD_TO_LREAL(DCH读遥控数据[5]);

DCH报警代码2 := LREAL_TO_INT(下桥SOC);
// IF 电量状态=0 THEN
// 	发动机启动 := TRUE;
// ELSIF 电量状态=2 THEN
// 	发动机启动 := FALSE;
// END_IF

DCH状态位.9 := DCH状态位_边沿2;
DCH状态位.10 := DCH状态位_边沿1;
DCH状态位.11 := DCH状态位_急停;
DCH状态位.12 := DCH状态位_报警;
DCH状态位.13 := DCH状态位_运行;
DCH状态位.14 := DCH状态位_手动;
DCH状态位.15 := DCH状态位_自动;

DCH写遥控数据[0] := DCH状态位;
DCH写遥控数据[1] := INT_TO_WORD(DCH报警代码1);
DCH写遥控数据[2] := INT_TO_WORD(DCH报警代码2);
DCH写遥控数据[3] := INT_TO_WORD(DCH上测距);
DCH写遥控数据[4] := INT_TO_WORD(DCH下测距);
END_METHOD

METHOD DCH底盘控制
VAR_INPUT
END_VAR
IF DCH电机控制0=FALSE THEN
	RETURN;
END_IF

IF DCH前进 OR DCH后退 OR DCH左转 OR DCH右转 THEN
	手动底盘联动 := TRUE;
	IF DCH前进 THEN
		手动左轮速度 := 底盘运行参数.底盘运行速度 * DCH前后数值量 / 255;
		手动右轮速度 := 底盘运行参数.底盘运行速度 * DCH前后数值量 / 255;
	END_IF
	IF DCH后退 THEN
		手动左轮速度 := 底盘运行参数.底盘运行速度 * DCH前后数值量 / 255 * -1;
		手动右轮速度 := 底盘运行参数.底盘运行速度 * DCH前后数值量 / 255 * -1;
	END_IF
	IF DCH左转 THEN
		手动左轮速度 := 手动左轮速度 - 底盘运行参数.底盘运行速度 * DCH左右数值量 / 255;
		手动右轮速度 := 手动右轮速度;
		IF 手动右轮速度=0 THEN
			手动右轮速度 := -手动左轮速度;
		END_IF
	END_IF
	IF DCH右转 THEN
		手动左轮速度 := 手动左轮速度;
		手动右轮速度 := 手动右轮速度 - 底盘运行参数.底盘运行速度 * DCH左右数值量 / 255;
		IF 手动左轮速度=0 THEN
			手动左轮速度 := -手动右轮速度;
		END_IF
	END_IF
ELSE
	手动左轮速度 := 0.0;
	手动右轮速度 := 0.0;
END_IF

IF DCH方向1正转 OR DCH方向1反转 THEN
	手动底盘联动 := FALSE;
	IF DCH方向1正转=TRUE THEN
		左上气缸伺服参数.运行模式 := 1;
		左上气缸伺服参数.运行方向 := TRUE;
	END_IF
	IF DCH方向1反转=TRUE THEN
		左上气缸伺服参数.运行模式 := 1;
		左上气缸伺服参数.运行方向 := FALSE;
	END_IF
ELSE
	左上气缸伺服参数.运行模式 := 0;
END_IF

IF DCH方向2正转 OR DCH方向2反转 THEN
	手动底盘联动 := FALSE;
	IF DCH方向2正转=TRUE THEN
		左下气缸伺服参数.运行模式 := 1;
		左下气缸伺服参数.运行方向 := TRUE;
	END_IF
	IF DCH方向2反转=TRUE THEN
		左下气缸伺服参数.运行模式 := 1;
		左下气缸伺服参数.运行方向 := FALSE;
	END_IF
ELSE
	左下气缸伺服参数.运行模式 := 0;
END_IF

IF DCH方向3正转 OR DCH方向3反转 THEN
	手动底盘联动 := FALSE;
	IF DCH方向3正转=TRUE THEN
		右上气缸伺服参数.运行模式 := 1;
		右上气缸伺服参数.运行方向 := TRUE;
	END_IF
	IF DCH方向3反转=TRUE THEN
		右上气缸伺服参数.运行模式 := 1;
		右上气缸伺服参数.运行方向 := FALSE;
	END_IF
ELSE
	右上气缸伺服参数.运行模式 := 0;
END_IF

IF DCH方向4正转 OR DCH方向4反转 THEN
	手动底盘联动 := FALSE;
	IF DCH方向4正转=TRUE THEN
		右下气缸伺服参数.运行模式 := 1;
		右下气缸伺服参数.运行方向 := TRUE;
	END_IF
	IF DCH方向4反转=TRUE THEN
		右下气缸伺服参数.运行模式 := 1;
		右下气缸伺服参数.运行方向 := FALSE;
	END_IF
ELSE
	右下气缸伺服参数.运行模式 := 0;
END_IF

// 	底盘运行参数.底盘运动方向 := SEL(DCH前进, 0, 1);
END_METHOD

METHOD DCH机械臂控制
VAR_INPUT
END_VAR
VAR
	运动触发标志	: BOOL;
END_VAR
//DCH机械臂控制
IF DCH电机控制1 OR DCH电机控制2 THEN
	IF DCH电机控制1=TRUE THEN
		机械臂运行参数.是否关节运动 := TRUE;
	END_IF
	IF DCH电机控制2=TRUE THEN
		机械臂运行参数.是否关节运动 := FALSE;
	END_IF
ELSE
	RETURN;
END_IF

IF DCH滚刷正转=TRUE THEN
	机械臂运行参数.倍率 := 90.0;
END_IF
IF DCH滚刷关闭=TRUE THEN
	机械臂运行参数.倍率 := 60.0;
END_IF
IF DCH滚刷反转=TRUE THEN
	机械臂运行参数.倍率 := 20.0;
END_IF

IF DCH方向1正转 OR DCH方向1反转 OR DCH方向2正转 OR DCH方向2反转 OR DCH方向3正转 OR DCH方向3反转 OR DCH方向4正转 OR DCH方向4反转 THEN
	IF 机械臂手动运行=FALSE THEN
		IF DCH方向1正转=TRUE THEN
			机械臂运行参数.轴号 := 0;
			机械臂运行参数.方向 := 1;
		END_IF
		IF DCH方向1反转=TRUE THEN
			机械臂运行参数.轴号 := 0;
			机械臂运行参数.方向 := 0;
		END_IF
		IF DCH方向2正转=TRUE THEN
			机械臂运行参数.轴号 := 1;
			机械臂运行参数.方向 := 1;
		END_IF
		IF DCH方向2反转=TRUE THEN
			机械臂运行参数.轴号 := 1;
			机械臂运行参数.方向 := 0;
		END_IF
		IF DCH方向3正转=TRUE THEN
			机械臂运行参数.轴号 := 2;
			机械臂运行参数.方向 := 1;
		END_IF
		IF DCH方向3反转=TRUE THEN
			机械臂运行参数.轴号 := 2;
			机械臂运行参数.方向 := 0;
		END_IF
		IF DCH方向4正转=TRUE THEN
			机械臂运行参数.轴号 := 3;
			机械臂运行参数.方向 := 1;
		END_IF
		IF DCH方向4反转=TRUE THEN
			机械臂运行参数.轴号 := 3;
			机械臂运行参数.方向 := 0;
		END_IF
		机械臂运行参数.规划模式 := 1;
		机械臂运行启动 := TRUE;
		机械臂手动运行 := TRUE;
	END_IF
ELSE
	IF 机械臂手动运行=TRUE THEN
		机械臂运行参数.规划模式 := 3;
		机械臂运行启动 := TRUE;
		机械臂手动运行 := FALSE;
	END_IF
END_IF

IF DCH启动=TRUE THEN
	机械臂运行参数.规划模式 := 4;
	机械臂运行参数.是否关节运动 := TRUE;
	机械臂运行参数.运行点位[0] := 0.0; 机械臂运行参数.运行点位[1] := -90.0; 机械臂运行参数.运行点位[2] := 180.0;
	机械臂运行参数.运行点位[3] := 45.0; 机械臂运行参数.运行点位[4] := 0.0; 机械臂运行参数.运行点位[5] := 0.0;
	IF sMotionOutputs.iRobStatus = 1 THEN
		机械臂运行启动 := TRUE;
	END_IF
END_IF

IF DCH停止=TRUE THEN
	机械臂运行参数.规划模式 := 5;
	IF sMotionOutputs.iRobStatus = 2 THEN
		机械臂运行启动 := TRUE;
	END_IF
END_IF
END_METHOD

END_PROGRAM

// Device/Application/SLAM指令通讯
PROGRAM SLAM指令通讯
VAR
	作业控制编码 : WORD;
	流程处理状态 : INT := 0;
	清扫返回状态 : BYTE;
	SktTCPSend_0: SktTCPSend;
	SktTCPRecv_0: SktTCPRecv;
	SktClose_0: SktClose;
	SktTCPGetStatus_0: SktTCPGetStatus;
	diConnectID: CONNECT_ID := 3;
	stServerAddress: ADDRESS;
	stConnectInfo: CONNECT_INFO;
	DataSend: ARRAY[0..1024] OF BYTE;
	DataRevice: ARRAY[0..1024] OF BYTE;
	start_tcp_communication: BOOL := FALSE;
	status: WORD := 0;
	R_TRIG_0: R_TRIG;
	F_TRIG_0: F_TRIG;
	start_tcp_server: BOOL;
	SktTCPServer_0: SktTCPServer;
	CanWR: BOOL;
	HandleDataRevice: ARRAY[0..2048] OF BYTE;
	NumRevc: WORD := 0;
	tmpRevc: WORD := 0;
	i: WORD := 0;
	校验功能块_0: 校验功能块;
	sumcheck: BYTE;
	SendSize: WORD;
	bSend: BOOL;
	tmpDataSend: ARRAY[0..200] OF BYTE;
	接收序列号: WORD;
	初始化: BOOL;
	TON_0: TON;
	TON_2: TON;
	bCloseSocket: BOOL := 0;
	上传信息处理_0: 上传信息处理;
	上传信息处理_1: 上传信息处理;
	上传信息处理_2: 上传信息处理;
	上传信息处理_3: 上传信息处理;
	上传信息处理_4: 上传信息处理;
	上传信息处理_5: 上传信息处理;
	上传信息处理_6: 上传信息处理;
	上传信息处理_7: 上传信息处理;
	上传信息处理_8: 上传信息处理;
	上传信息处理_9: 上传信息处理;
END_VAR

R_TRIG_0(CLK:=SLAM通讯复位 , Q=> );
F_TRIG_0(CLK:=SLAM通讯复位 , Q=> );

TON_0(IN:=自动重连 AND status = 255 , PT:=T#1S , Q=> , ET=> );
TON_2(IN:=SktClose_0.xExecute AND status = 4 , PT:=T#3S , Q=> , ET=> );
IF TON_2.Q THEN
	status := 1;
	SktClose_0(xExecute:=FALSE);		
	SktTCPGetStatus_0(xEnable:=FALSE);
	start_tcp_server := FALSE;	
	CanWR := 0;
	NumRevc :=0;
	SLAM连接状态 := 0;
	bSend := 0;
	bCloseSocket := 0;
END_IF


IF F_TRIG_0.Q OR NOT 初始化 OR TON_0.Q THEN
	status := 1;
END_IF
IF   R_TRIG_0.Q  THEN 
	IF status=1 THEN
		status := 255;
	ELSIF status=2 THEN
		status := 255;
	ELSIF status=3 THEN
		status := 4;
	END_IF	
END_IF

SktTCPServer_0(
		xExecute:= start_tcp_server, 
		diConnectID:= diConnectID, 
		strLocalAddress:= stServerAddress, 
		xDone=> , 
		xBusy=> , 
		xError=> , 
		wErrorID=> , 
		stConnectInfo=> stConnectInfo);

SktClose_0(
		xExecute:= bCloseSocket, 
		diConnectID:=stConnectInfo.diConnectID ,
		xDone=> ,
		xBusy=> ,
		xError=> ,
		wErrorID=> );


CASE status OF
	1:
		SLAM连接状态 := 0;
		stServerAddress.strIPAddr := '0.0.0.0';
		stServerAddress.uiPort := 8000;
		//diConnectID := 3;
		start_tcp_server := TRUE;
		status := 2;
		CanWR := 0;
		bCloseSocket := 0;

	2:		
		IF SktTCPServer_0.xDone THEN
			status := 3;
			JMP RUN_RND;			
		ELSIF SktTCPServer_0.xError THEN		
			IF SktTCPServer_0.wErrorID = 21 THEN
				IF diConnectID <50 THEN
					diConnectID := diConnectID +1;
				ELSE
					diConnectID := 3;
				END_IF
				
			ELSE
				status := 255;
			END_IF
					
			JMP RUN_RND;
		END_IF
	3:
		CanWR := 0;
		SktTCPGetStatus_0(
			xEnable:= TRUE, 
			diConnectID:= stConnectInfo.diConnectID, 
			xDone=> , 
			xBusy=> , 
			xError=> , 
			wErrorID=> , 
			eStatus=> , 
			stConnectInfo=> );
		IF SktTCPGetStatus_0.xError THEN
			status := 4;
			SLAM连接状态 := 0;
			JMP RUN_RND;
		ELSIF SktTCPGetStatus_0.eStatus <> CmpHCTCPIP.TCP_STATUS.TCP_ESTABLISHED THEN
			status := 4;
			SLAM连接状态 := 0;
			JMP RUN_RND;
			;
		ELSE
			SLAM连接状态 := 1;
			CanWR := 1;
		END_IF
	
	4:
		bCloseSocket := 1;
		IF SktClose_0.xDone THEN
			status := 255;
			JMP RUN_RND;
		END_IF
		CanWR :=0;
	255:
		bCloseSocket := 0;		
		SktTCPGetStatus_0(xEnable:=FALSE);
		//SktTCPServer_0(xExecute:= FALSE);
		start_tcp_server := FALSE;	
		CanWR := 0;
		NumRevc :=0;
		SLAM连接状态 := 0;
		bSend := 0;
END_CASE

SktTCPRecv_0(
	xEnable:= CanWR, 
	diConnectID:= stConnectInfo.diConnectID, 
	abyData:= DataRevice[0], 
	uiDataSize:= 0, 
	xDone=> , 
	xBusy=> , 
	xError=> , 
	wErrorID=> , 
	xReady=> , 
	uiCount=> );
IF SktTCPRecv_0.xError THEN
	status := 4;
	JMP RUN_RND;
ELSIF SktTCPRecv_0.xDone AND NOT(SktTCPRecv_0.xError) THEN
	status := 255;
	JMP RUN_RND;
ELSE
	IF SktTCPRecv_0.xReady THEN
		tmpRevc := 0;
		IF (2048-NumRevc) < SktTCPRecv_0.uiCount THEN
			tmpRevc := SktTCPRecv_0.uiCount - (2048-NumRevc);					
		END_IF
		AryMove(In:=DataRevice[0] , AryOut:=HandleDataRevice[NumRevc] , Size:=SktTCPRecv_0.uiCount - tmpRevc );	
		NumRevc := NumRevc + SktTCPRecv_0.uiCount - tmpRevc;
	END_IF	
END_IF
tmpRevc := 0;

IF NumRevc >= 7 AND NumRevc <2048 THEN
	FOR i:=0 TO NumRevc-1 BY 1 DO
		IF HandleDataRevice[i] =  16#5A THEN
			IF (NumRevc -i) >=7 THEN
				IF HandleDataRevice[i+1] = 16#A5 THEN
					IF (i+HandleDataRevice[i+2]+2) <= NumRevc THEN
						校验功能块_0(pData:=ADR(HandleDataRevice[i]), sizeNome:=HandleDataRevice[i+2]+1 , sumCheck=>sumcheck );
						IF HandleDataRevice[HandleDataRevice[i+2]+1+i] = sumcheck  THEN // 处理
							CASE HandleDataRevice[i+5] OF
								16#00:
									IF HandleDataRevice[i+6] = 16#00 THEN
										IF HandleDataRevice[i+7] = 0  THEN
											SLAM急停 := 0;
										ELSE
											SLAM急停 := 1;
										END_IF
										接收序列号 := SHL(BYTE_TO_WORD( HandleDataRevice[i+4]), 8) OR HandleDataRevice[i+5];
										上传信息处理_0(定时时间 :=T#0S , 数据域长度 := 0,  pInputData := , 应答 :=16#00 , 序列号 :=接收序列号 , 主功能码 :=16#00 , 次功能码 :=16#00 );
									END_IF								
								16#01:
									IF HandleDataRevice[i+6] = 16#00 THEN
										// 千寻传输的Vx、Vy、Wz的值因浮点数传输的关系扩大了100倍，实际数值需除100
										Vx := WORD_TO_INT(SHL(BYTE_TO_WORD(HandleDataRevice[i+7]), 8) OR HandleDataRevice[i+8]);
										Vy := WORD_TO_INT(SHL(BYTE_TO_WORD(HandleDataRevice[i+9]), 8) OR HandleDataRevice[i+10]);
										Wz := WORD_TO_INT(SHL(BYTE_TO_WORD(HandleDataRevice[i+11]), 8) OR HandleDataRevice[i+12]);	// 单位为弧度/s
										SLAM左轮速度 := (INT_TO_LREAL(Vx)/100.0 - (INT_TO_LREAL(Wz)/100.0 * 1.6935) / 2) * 1000.0; // 转换为毫米/s下发至伺服，dVelFac为实验数据所得
										SLAM右轮速度 := (INT_TO_LREAL(Vx)/100.0 + (INT_TO_LREAL(Wz)/100.0 * 1.6935) / 2) * 1000.0;
										SLAM速度有效 := TRUE;
										IF HandleDataRevice[i+14] = 0 THEN
											SLAM控制方式 := 0;
										ELSE
											SLAM控制方式 := 1;
										END_IF
										接收序列号 := SHL(BYTE_TO_WORD( HandleDataRevice[i+3]), 8) OR HandleDataRevice[i+4];
										上传信息处理_0(定时时间:=T#0MS, 数据域长度:= 0, 应答:= 16#00, 序列号:=接收序列号, 主功能码:= 16#01, 次功能码:= 16#00);
									END_IF
							END_CASE
                            i := i + HandleDataRevice[i+2]+1;
							tmpRevc := i+1;
						END_IF
					ELSE
						JMP RUN_ENDFOR;
					END_IF
				ELSE
					tmpRevc := tmpRevc +1;
				END_IF
			ELSE
				JMP RUN_ENDFOR;
			END_IF
		ELSE
			tmpRevc := tmpRevc +1;
		END_IF;
	END_FOR
END_IF

RUN_ENDFOR:
IF tmpRevc > 0 THEN
	ArySHR(InOut:=HandleDataRevice[0] , Size:=2048 , Num:=tmpRevc );
	NumRevc := NumRevc - tmpRevc;
END_IF


{region}//上传

IF CanWR THEN
// 	系统状态上传();
	轮速计数据上传();
// 	BMS数据上传();
// 	UPS数据上传();
// 	单体电池电压数据上传(电池组序号:=0);
// 	单体电池电压数据上传(电池组序号:=1);
// 	单体电池电压数据上传(电池组序号:=2);
// 	单体电池电压数据上传(电池组序号:=3);
// 	单体电池温度数据上传(循环时间:=T#9950MS, 电池组序号:=0);
// 	单体电池温度数据上传(循环时间:=T#9900MS, 电池组序号:=1);
// 	单体电池温度数据上传(循环时间:=T#9850MS, 电池组序号:=2);
// 	单体电池温度数据上传(循环时间:=T#9800MS, 电池组序号:=3);
// 	行走电机状态上传();
// 	悬挂电机状态上传();
// 	超声波数据上传();

END_IF
{end}{	{region}

IF 待发送缓存数组长度 >0 AND bSend = 0 THEN
	SendSize := 待发送缓存数组长度;
	AryMove(In:=待发送缓存数组[0] , AryOut:=DataSend[0] , Size:= SendSize);
	待发送缓存数组长度 :=0;
	bSend := 1;
END_IF
SktTCPSend_0(
	xExecute:= bSend, 
	diConnectID:= stConnectInfo.diConnectID, 
	abyData:= DataSend[0], 
	uiDataSize:= SendSize, 
	uiTimeOut:= 500, 
	xDone=> , 
	xBusy=> , 
	xError=> , 
	wErrorID=> );
IF SktTCPSend_0.xError THEN
	status := 4;
	JMP RUN_RND;
ELSIF SktTCPSend_0.xDone THEN
	bSend := 0; //发送完毕
	SendSize := 0;
END_IF


RUN_RND:

//SLAM通讯不上 := NOT SLAM连接状态;
IF NOT 初始化 THEN
	初始化 :=1;
// 	// 每 20 s 刷新一次（其实只在第一次扫描时执行一次）
//     FOR i := 1 TO 16 DO
//         ProbeTemp[i] := BYTE(50 + i MOD 20);   // 50..69 → 0..19 ℃
//     END_FOR
END_IF

METHOD 系统状态上传
VAR_INPUT
END_VAR
//系统状态 [0x04,0x00]
tmpDataSend[0] := 16#00;
tmpDataSend[1] := 16#01;
tmpDataSend[2] := 16#00; //遥控器信号强度
tmpDataSend[3] := 16#00; //0-正常 1-急停
tmpDataSend[4] := 16#00;
tmpDataSend[5] := 16#00;
tmpDataSend[6] := 16#00;
tmpDataSend[7] := 16#00;

上传信息处理_6(定时时间:=T#500MS, 数据域长度:=8, pInputData:=ADR(tmpDataSend[0]), 应答:=16#00, 序列号:=上传序列号, 主功能码:=16#04, 次功能码:=16#00);
END_METHOD

METHOD BMS数据上传
VAR_INPUT
END_VAR
VAR
END_VAR
//2.4.8 BMS数据 [0x04,0x07]
tmpDataSend[0] := WORD_TO_BYTE(BMS映射数据[0]); // 系统状态: 0-初始化 1-待机模式 2-充电模式 3-放电模式 4-上电BCU编码中 5-上电BMU编码中 6-上电绝缘检测中 7-上电并机中 8-掉电中 9-系统锁定
tmpDataSend[1] := WORD_TO_BYTE(BMS映射数据[1]);  // 电池状态: 0-等待 1-禁充禁放 2-禁充 3-禁放 4-充电中 5-放电中

// 三级保护 
//一级保护状态
tmpDataSend[2] := WORD_TO_BYTE(SHR(BMS映射数据[2], 8));
tmpDataSend[3] := WORD_TO_BYTE(BMS映射数据[2] AND 16#FF);
tmpDataSend[4] := WORD_TO_BYTE(SHR(BMS映射数据[3], 8));
tmpDataSend[5] := WORD_TO_BYTE(BMS映射数据[3] AND 16#FF);
//二级保护状态
tmpDataSend[6] := WORD_TO_BYTE(SHR(BMS映射数据[4], 8));
tmpDataSend[7] := WORD_TO_BYTE(BMS映射数据[4] AND 16#FF);
tmpDataSend[8] := WORD_TO_BYTE(SHR(BMS映射数据[5], 8));
tmpDataSend[9] := WORD_TO_BYTE(BMS映射数据[5] AND 16#FF);
//三级保护状态
tmpDataSend[10] := WORD_TO_BYTE(SHR(BMS映射数据[6], 8));
tmpDataSend[11] := WORD_TO_BYTE(BMS映射数据[6] AND 16#FF);
tmpDataSend[12] := WORD_TO_BYTE(SHR(BMS映射数据[7], 8));
tmpDataSend[13] := WORD_TO_BYTE(BMS映射数据[7] AND 16#FF);

// 故障状态 2 字节
tmpDataSend[14] := WORD_TO_BYTE(SHR(BMS映射数据[8], 8));
tmpDataSend[15] := WORD_TO_BYTE(BMS映射数据[8] AND 16#FF);
tmpDataSend[16] := WORD_TO_BYTE(SHR(BMS映射数据[9], 8));
tmpDataSend[17] := WORD_TO_BYTE(BMS映射数据[9] AND 16#FF);

// 2) 电压 & 电流 
// 采集电压        
tmpDataSend[18] := WORD_TO_BYTE(SHR(BMS映射数据[10], 8)); 	// 0.1V
tmpDataSend[19] := WORD_TO_BYTE(BMS映射数据[10] AND 16#FF);

// 负载电压  
tmpDataSend[20] := WORD_TO_BYTE(SHR(BMS映射数据[11], 8));		// 0.1V
tmpDataSend[21] := WORD_TO_BYTE(BMS映射数据[11] AND 16#FF);

// 上桥累计电压 
tmpDataSend[22] := WORD_TO_BYTE(SHR(BMS映射数据[12], 8));		// 0.1V
tmpDataSend[23] := WORD_TO_BYTE(BMS映射数据[12] AND 16#FF);

// 下桥累计电压
tmpDataSend[24] := WORD_TO_BYTE(SHR(BMS映射数据[13], 8));		// 0.1V
tmpDataSend[25] := WORD_TO_BYTE(BMS映射数据[13] AND 16#FF);

// 上桥电流
tmpDataSend[26] := WORD_TO_BYTE(SHR(BMS映射数据[14], 8));		// 0.01A
tmpDataSend[27] := WORD_TO_BYTE(BMS映射数据[14] AND 16#FF);
tmpDataSend[28] := WORD_TO_BYTE(SHR(BMS映射数据[15], 8));
tmpDataSend[29] := WORD_TO_BYTE(BMS映射数据[15] AND 16#FF);

//下桥电流
tmpDataSend[30] := WORD_TO_BYTE(SHR(BMS映射数据[16], 8));		// 0.01A
tmpDataSend[31] := WORD_TO_BYTE(BMS映射数据[16] AND 16#FF);
tmpDataSend[32] := WORD_TO_BYTE(SHR(BMS映射数据[17], 8));
tmpDataSend[33] := WORD_TO_BYTE(BMS映射数据[17] AND 16#FF);

// 上/下桥SOC 
tmpDataSend[34] := WORD_TO_BYTE(BMS映射数据[18]);		// %
tmpDataSend[35] := WORD_TO_BYTE(BMS映射数据[19]);	

// 上/下桥SOH
tmpDataSend[36] := WORD_TO_BYTE(BMS映射数据[20]);		// %
tmpDataSend[37] := WORD_TO_BYTE(BMS映射数据[21]);	

// 上/下桥电池剩余容量
tmpDataSend[38] := WORD_TO_BYTE(SHR(BMS映射数据[22], 8));	
tmpDataSend[39] := WORD_TO_BYTE(BMS映射数据[22] AND 16#FF);
tmpDataSend[40] := WORD_TO_BYTE(SHR(BMS映射数据[23], 8));	
tmpDataSend[41] := WORD_TO_BYTE(BMS映射数据[23] AND 16#FF);

tmpDataSend[42] := WORD_TO_BYTE(SHR(BMS映射数据[24], 8));	
tmpDataSend[43] := WORD_TO_BYTE(BMS映射数据[24] AND 16#FF);
tmpDataSend[44] := WORD_TO_BYTE(SHR(BMS映射数据[25], 8));	
tmpDataSend[45] := WORD_TO_BYTE(BMS映射数据[25] AND 16#FF);

// 上/下桥功率百分比
tmpDataSend[46] := WORD_TO_BYTE(SHR(BMS映射数据[26], 8));		// 0.1KW
tmpDataSend[47] := WORD_TO_BYTE(BMS映射数据[26] AND 16#FF);
tmpDataSend[48] := WORD_TO_BYTE(SHR(BMS映射数据[27], 8));		// 0.1KW
tmpDataSend[49] := WORD_TO_BYTE(BMS映射数据[27] AND 16#FF);

// 周期 10 s，固定 48 Byte
上传信息处理_5(定时时间:=T#9990MS, 数据域长度:=50, pInputData:=ADR(tmpDataSend[0]), 应答:=16#00, 序列号:=上传序列号, 主功能码:=16#04, 次功能码:=16#07);
END_METHOD

METHOD 温湿度数据上传
VAR_INPUT
END_VAR
//温湿度数据 [0x04,0x08]
tmpDataSend[0] := 16#00;
tmpDataSend[1] := 16#01;
tmpDataSend[2] := 16#00; //遥控器信号强度
tmpDataSend[3] := 16#00; //0-正常 1-急停
tmpDataSend[4] := 16#00;
tmpDataSend[5] := 16#00;
tmpDataSend[6] := 16#00;
tmpDataSend[7] := 16#00;

上传信息处理_6(定时时间:=T#10000MS, 数据域长度:=8, pInputData:=ADR(tmpDataSend[0]), 应答:=16#00, 序列号:=上传序列号, 主功能码:=16#04, 次功能码:=16#08);
END_METHOD

METHOD 单体电池电压数据上传
VAR_INPUT
	电池组序号	 : INT;
END_VAR
VAR
	iCounter	 : INT;
	电池电压组缓存 : ARRAY [0..29] OF WORD;
END_VAR
FOR iCounter:=0 TO 29 BY 1 DO
	电池电压组缓存[iCounter] := 电池映射电压组1[iCounter];
END_FOR

tmpDataSend[0] := WORD_TO_BYTE(BMS映射数据[1]);  // 电池状态: 0-等待 1-禁充禁放 2-禁充 3-禁放 4-充电中 5-放电中
tmpDataSend[1] := INT_TO_BYTE(电池组序号);
tmpDataSend[2] := WORD_TO_BYTE(SHR(电池电压组缓存[0], 8));	//0.001V
tmpDataSend[3] := WORD_TO_BYTE(电池电压组缓存[0] AND 16#FF);
tmpDataSend[4] := WORD_TO_BYTE(SHR(电池电压组缓存[1], 8));
tmpDataSend[5] := WORD_TO_BYTE(电池电压组缓存[1] AND 16#FF);
tmpDataSend[6] := WORD_TO_BYTE(SHR(电池电压组缓存[2], 8));
tmpDataSend[7] := WORD_TO_BYTE(电池电压组缓存[2] AND 16#FF);
tmpDataSend[8] := WORD_TO_BYTE(SHR(电池电压组缓存[3], 8));
tmpDataSend[9] := WORD_TO_BYTE(电池电压组缓存[3] AND 16#FF);
tmpDataSend[10] := WORD_TO_BYTE(SHR(电池电压组缓存[4], 8));
tmpDataSend[11] := WORD_TO_BYTE(电池电压组缓存[4] AND 16#FF);
tmpDataSend[12] := WORD_TO_BYTE(SHR(电池电压组缓存[5], 8));
tmpDataSend[13] := WORD_TO_BYTE(电池电压组缓存[5] AND 16#FF);
tmpDataSend[14] := WORD_TO_BYTE(SHR(电池电压组缓存[6], 8));
tmpDataSend[15] := WORD_TO_BYTE(电池电压组缓存[6] AND 16#FF);
tmpDataSend[16] := WORD_TO_BYTE(SHR(电池电压组缓存[7], 8));
tmpDataSend[17] := WORD_TO_BYTE(电池电压组缓存[7] AND 16#FF);     
tmpDataSend[18] := WORD_TO_BYTE(SHR(电池电压组缓存[8], 8));
tmpDataSend[19] := WORD_TO_BYTE(电池电压组缓存[8] AND 16#FF);
tmpDataSend[20] := WORD_TO_BYTE(SHR(电池电压组缓存[9], 8));
tmpDataSend[21] := WORD_TO_BYTE(电池电压组缓存[9] AND 16#FF);
tmpDataSend[22] := WORD_TO_BYTE(SHR(电池电压组缓存[10], 8));
tmpDataSend[23] := WORD_TO_BYTE(电池电压组缓存[10] AND 16#FF);
tmpDataSend[24] := WORD_TO_BYTE(SHR(电池电压组缓存[11], 8));
tmpDataSend[25] := WORD_TO_BYTE(电池电压组缓存[11] AND 16#FF);
tmpDataSend[26] := WORD_TO_BYTE(SHR(电池电压组缓存[12], 8));
tmpDataSend[27] := WORD_TO_BYTE(电池电压组缓存[12] AND 16#FF);
tmpDataSend[28] := WORD_TO_BYTE(SHR(电池电压组缓存[13], 8));
tmpDataSend[29] := WORD_TO_BYTE(电池电压组缓存[13] AND 16#FF);
tmpDataSend[30] := WORD_TO_BYTE(SHR(电池电压组缓存[14], 8));
tmpDataSend[31] := WORD_TO_BYTE(电池电压组缓存[14] AND 16#FF);
tmpDataSend[32] := WORD_TO_BYTE(SHR(电池电压组缓存[15], 8));
tmpDataSend[33] := WORD_TO_BYTE(电池电压组缓存[15] AND 16#FF);
tmpDataSend[34] := WORD_TO_BYTE(SHR(电池电压组缓存[16], 8));
tmpDataSend[35] := WORD_TO_BYTE(电池电压组缓存[16] AND 16#FF);
tmpDataSend[36] := WORD_TO_BYTE(SHR(电池电压组缓存[17], 8));
tmpDataSend[37] := WORD_TO_BYTE(电池电压组缓存[17] AND 16#FF);
tmpDataSend[38] := WORD_TO_BYTE(SHR(电池电压组缓存[18], 8));	
tmpDataSend[39] := WORD_TO_BYTE(电池电压组缓存[18] AND 16#FF);
tmpDataSend[40] := WORD_TO_BYTE(SHR(电池电压组缓存[19], 8));	
tmpDataSend[41] := WORD_TO_BYTE(电池电压组缓存[19] AND 16#FF);
tmpDataSend[42] := WORD_TO_BYTE(SHR(电池电压组缓存[20], 8));	
tmpDataSend[43] := WORD_TO_BYTE(电池电压组缓存[20] AND 16#FF);
tmpDataSend[44] := WORD_TO_BYTE(SHR(电池电压组缓存[21], 8));	
tmpDataSend[45] := WORD_TO_BYTE(电池电压组缓存[21] AND 16#FF);
tmpDataSend[46] := WORD_TO_BYTE(SHR(电池电压组缓存[22], 8));
tmpDataSend[47] := WORD_TO_BYTE(电池电压组缓存[22] AND 16#FF);
tmpDataSend[48] := WORD_TO_BYTE(SHR(电池电压组缓存[23], 8));
tmpDataSend[49] := WORD_TO_BYTE(电池电压组缓存[23] AND 16#FF);
tmpDataSend[50] := WORD_TO_BYTE(SHR(电池电压组缓存[24], 8));
tmpDataSend[51] := WORD_TO_BYTE(电池电压组缓存[24] AND 16#FF);
tmpDataSend[52] := WORD_TO_BYTE(SHR(电池电压组缓存[25], 8));
tmpDataSend[53] := WORD_TO_BYTE(电池电压组缓存[25] AND 16#FF);
tmpDataSend[54] := WORD_TO_BYTE(SHR(电池电压组缓存[26], 8));
tmpDataSend[55] := WORD_TO_BYTE(电池电压组缓存[26] AND 16#FF);
tmpDataSend[56] := WORD_TO_BYTE(SHR(电池电压组缓存[27], 8));
tmpDataSend[57] := WORD_TO_BYTE(电池电压组缓存[27] AND 16#FF);
tmpDataSend[58] := WORD_TO_BYTE(SHR(电池电压组缓存[28], 8));
tmpDataSend[59] := WORD_TO_BYTE(电池电压组缓存[28] AND 16#FF);
tmpDataSend[60] := WORD_TO_BYTE(SHR(电池电压组缓存[29], 8));
tmpDataSend[61] := WORD_TO_BYTE(电池电压组缓存[29] AND 16#FF);

上传信息处理_9(定时时间:=T#9960MS, 数据域长度:=62, pInputData:=ADR(tmpDataSend[0]), 应答:=16#00, 序列号:=上传序列号, 主功能码:=16#04, 次功能码:=16#08);
END_METHOD

METHOD 单体电池温度数据上传
VAR_INPUT
	电池组序号	: INT;
	循环时间		: TIME;
END_VAR
VAR
	iCounter	 : INT;
	电池温度组缓存 : ARRAY [0..9] OF WORD;
	上传信息处理调用	: 上传信息处理;
END_VAR
FOR iCounter:=0 TO 9 BY 1 DO
	电池温度组缓存[iCounter] := 电池映射温度组1[iCounter];
END_FOR

tmpDataSend[0] := INT_TO_BYTE(电池组序号);
tmpDataSend[1] := WORD_TO_BYTE(SHR(电池温度组缓存[0], 8));	//0.1度
tmpDataSend[2] := WORD_TO_BYTE(电池温度组缓存[0] AND 16#FF);
tmpDataSend[3] := WORD_TO_BYTE(SHR(电池温度组缓存[1], 8));
tmpDataSend[4] := WORD_TO_BYTE(电池温度组缓存[1] AND 16#FF);
tmpDataSend[5] := WORD_TO_BYTE(SHR(电池温度组缓存[2], 8));
tmpDataSend[6] := WORD_TO_BYTE(电池温度组缓存[2] AND 16#FF);
tmpDataSend[7] := WORD_TO_BYTE(SHR(电池温度组缓存[3], 8));
tmpDataSend[8] := WORD_TO_BYTE(电池温度组缓存[3] AND 16#FF);
tmpDataSend[9] := WORD_TO_BYTE(SHR(电池温度组缓存[4], 8));
tmpDataSend[10] := WORD_TO_BYTE(电池温度组缓存[4] AND 16#FF);
tmpDataSend[11] := WORD_TO_BYTE(SHR(电池温度组缓存[5], 8));
tmpDataSend[12] := WORD_TO_BYTE(电池温度组缓存[5] AND 16#FF);
tmpDataSend[13] := WORD_TO_BYTE(SHR(电池温度组缓存[6], 8));
tmpDataSend[14] := WORD_TO_BYTE(电池温度组缓存[6] AND 16#FF);
tmpDataSend[15] := WORD_TO_BYTE(SHR(电池温度组缓存[7], 8));
tmpDataSend[16] := WORD_TO_BYTE(电池温度组缓存[7] AND 16#FF);
tmpDataSend[17] := WORD_TO_BYTE(SHR(电池温度组缓存[8], 8));
tmpDataSend[18] := WORD_TO_BYTE(电池温度组缓存[8] AND 16#FF);
tmpDataSend[19] := WORD_TO_BYTE(SHR(电池温度组缓存[9], 8));
tmpDataSend[20] := WORD_TO_BYTE(电池温度组缓存[9] AND 16#FF);

上传信息处理_8(定时时间:=循环时间, 数据域长度:=21, pInputData:=ADR(tmpDataSend[0]), 应答:=16#00, 序列号:=上传序列号, 主功能码:=16#04, 次功能码:=16#09);
// 上传信息处理调用(定时时间:=循环时间, 数据域长度:=21, pInputData:=ADR(tmpDataSend[0]), 应答:=16#00, 序列号:=上传序列号, 主功能码:=16#04, 次功能码:=16#09);
END_METHOD

METHOD 行走电机状态上传
VAR_INPUT
END_VAR
VAR
	左上轮伺服电流	: WORD;
	左上轮伺服温度	: WORD;
	左上轮伺服报错码	: WORD;
	左下轮伺服电流	: WORD;
	左下轮伺服温度	: WORD;
	左下轮伺服报错码	: WORD;
	
	右上轮伺服电流	: WORD;
	右上轮伺服温度	: WORD;
	右上轮伺服报错码	: WORD;
	右下轮伺服电流	: WORD;
	右下轮伺服温度	: WORD;
	右下轮伺服报错码	: WORD;
END_VAR
//行走电机数据 [0x04,0x01]
左上轮伺服电流 := LREAL_TO_WORD(左上轮伺服参数.反馈电流);
左上轮伺服温度 := LREAL_TO_WORD(37);
左上轮伺服报错码 := LREAL_TO_WORD(0);
左下轮伺服电流 := LREAL_TO_WORD(左下轮伺服参数.反馈电流);
左下轮伺服温度 := LREAL_TO_WORD(37);
左下轮伺服报错码 := LREAL_TO_WORD(0);
右上轮伺服电流 := LREAL_TO_WORD(右上轮伺服参数.反馈电流);
右上轮伺服温度 := LREAL_TO_WORD(37);
右上轮伺服报错码 := LREAL_TO_WORD(0);
右下轮伺服电流 := LREAL_TO_WORD(右下轮伺服参数.反馈电流);
右下轮伺服温度 := LREAL_TO_WORD(37);
右下轮伺服报错码 := LREAL_TO_WORD(0);

tmpDataSend[0] := WORD_TO_BYTE(SHR(左上轮伺服电流, 8));
tmpDataSend[1] := WORD_TO_BYTE(左上轮伺服电流 AND 16#FF);
tmpDataSend[2] := WORD_TO_BYTE(SHR(左上轮伺服温度, 8));
tmpDataSend[3] := WORD_TO_BYTE(左上轮伺服温度 AND 16#FF);
tmpDataSend[4] := WORD_TO_BYTE(SHR(左上轮伺服报错码, 8));
tmpDataSend[5] := WORD_TO_BYTE(左上轮伺服报错码 AND 16#FF);
tmpDataSend[6] := 16#01;	//0-离线 1-在线

tmpDataSend[7] := WORD_TO_BYTE(SHR(左下轮伺服电流, 8));
tmpDataSend[8] := WORD_TO_BYTE(左下轮伺服电流 AND 16#FF);
tmpDataSend[9] := WORD_TO_BYTE(SHR(左下轮伺服温度, 8));
tmpDataSend[10] := WORD_TO_BYTE(左下轮伺服温度 AND 16#FF);
tmpDataSend[11] := WORD_TO_BYTE(SHR(左下轮伺服报错码, 8));
tmpDataSend[12] := WORD_TO_BYTE(左下轮伺服报错码 AND 16#FF);
tmpDataSend[13] := 16#01;	//0-离线 1-在线

tmpDataSend[14] := WORD_TO_BYTE(SHR(右上轮伺服电流, 8));
tmpDataSend[15] := WORD_TO_BYTE(右上轮伺服电流 AND 16#FF);
tmpDataSend[16] := WORD_TO_BYTE(SHR(右上轮伺服温度, 8));
tmpDataSend[17] := WORD_TO_BYTE(右上轮伺服温度 AND 16#FF);
tmpDataSend[18] := WORD_TO_BYTE(SHR(右上轮伺服报错码, 8));
tmpDataSend[19] := WORD_TO_BYTE(右上轮伺服报错码 AND 16#FF);
tmpDataSend[20] := 16#01;	//0-离线 1-在线

tmpDataSend[21] := WORD_TO_BYTE(SHR(右下轮伺服电流, 8));
tmpDataSend[22] := WORD_TO_BYTE(右下轮伺服电流 AND 16#FF);
tmpDataSend[23] := WORD_TO_BYTE(SHR(右下轮伺服温度, 8));
tmpDataSend[24] := WORD_TO_BYTE(右下轮伺服温度 AND 16#FF);
tmpDataSend[25] := WORD_TO_BYTE(SHR(右下轮伺服报错码, 8));
tmpDataSend[26] := WORD_TO_BYTE(右下轮伺服报错码 AND 16#FF);
tmpDataSend[27] := 16#01;	//0-离线 1-在线

上传信息处理_4(定时时间:=T#1000MS, 数据域长度:=28, pInputData:=ADR(tmpDataSend[0]), 应答:=16#00, 序列号:=上传序列号, 主功能码:=16#04, 次功能码:=16#01);
END_METHOD

METHOD 悬挂电机状态上传
VAR_INPUT
END_VAR
VAR
	左上悬挂伺服电流	: WORD;
	左上悬挂伺服位置	: WORD;
	左上悬挂伺服速度	: WORD;
	左上悬挂伺服温度	: WORD;
	左上悬挂伺服报错码	: WORD;
	左下悬挂伺服电流	: WORD;
	左下悬挂伺服位置	: WORD;
	左下悬挂伺服速度	: WORD;
	左下悬挂伺服温度	: WORD;
	左下悬挂伺服报错码	: WORD;
	
	右上悬挂伺服电流	: WORD;
	右上悬挂伺服位置	: WORD;
	右上悬挂伺服速度	: WORD;
	右上悬挂伺服温度	: WORD;
	右上悬挂伺服报错码	: WORD;
	右下悬挂伺服电流	: WORD;
	右下悬挂伺服位置	: WORD;
	右下悬挂伺服速度	: WORD;
	右下悬挂伺服温度	: WORD;
	右下悬挂伺服报错码	: WORD;
END_VAR
//悬挂电机数据 [0x04,0x02]
左上悬挂伺服电流 := LREAL_TO_WORD(左上气缸伺服参数.反馈电流);
左上悬挂伺服位置 := LREAL_TO_WORD(左上气缸伺服参数.反馈位置);
左上悬挂伺服速度 := LREAL_TO_WORD(左上气缸伺服参数.反馈速度);
左上悬挂伺服温度 := LREAL_TO_WORD(37);
左上悬挂伺服报错码 := LREAL_TO_WORD(0);
左下悬挂伺服电流 := LREAL_TO_WORD(左下气缸伺服参数.反馈电流);
左下悬挂伺服位置 := LREAL_TO_WORD(左下气缸伺服参数.反馈位置);
左下悬挂伺服速度 := LREAL_TO_WORD(左下气缸伺服参数.反馈速度);
左下悬挂伺服温度 := LREAL_TO_WORD(37);
左下悬挂伺服报错码 := LREAL_TO_WORD(0);

右上悬挂伺服电流 := LREAL_TO_WORD(右上气缸伺服参数.反馈电流);
右上悬挂伺服位置 := LREAL_TO_WORD(右上气缸伺服参数.反馈位置);
右上悬挂伺服速度 := LREAL_TO_WORD(右上气缸伺服参数.反馈速度);
右上悬挂伺服温度 := LREAL_TO_WORD(37);
右上悬挂伺服报错码 := LREAL_TO_WORD(0);
右下悬挂伺服电流 := LREAL_TO_WORD(右下气缸伺服参数.反馈电流);
右下悬挂伺服位置 := LREAL_TO_WORD(右下气缸伺服参数.反馈位置);
右下悬挂伺服速度 := LREAL_TO_WORD(右下气缸伺服参数.反馈速度);
右下悬挂伺服温度 := LREAL_TO_WORD(37);
右下悬挂伺服报错码 := LREAL_TO_WORD(0);

tmpDataSend[0] := WORD_TO_BYTE(SHR(左上悬挂伺服电流, 8));
tmpDataSend[1] := WORD_TO_BYTE(左上悬挂伺服电流 AND 16#FF);
tmpDataSend[2] := WORD_TO_BYTE(SHR(左上悬挂伺服位置, 8));
tmpDataSend[3] := WORD_TO_BYTE(左上悬挂伺服位置 AND 16#FF);
tmpDataSend[4] := WORD_TO_BYTE(SHR(左上悬挂伺服速度, 8));
tmpDataSend[5] := WORD_TO_BYTE(左上悬挂伺服速度 AND 16#FF);
tmpDataSend[6] := WORD_TO_BYTE(SHR(左上悬挂伺服温度, 8));
tmpDataSend[7] := WORD_TO_BYTE(左上悬挂伺服温度 AND 16#FF);
tmpDataSend[8] := WORD_TO_BYTE(SHR(左上悬挂伺服报错码, 8));
tmpDataSend[9] := WORD_TO_BYTE(左上悬挂伺服报错码 AND 16#FF);
tmpDataSend[10] := 16#01;	//0-离线 1-在线

tmpDataSend[11] := WORD_TO_BYTE(SHR(左下悬挂伺服电流, 8));
tmpDataSend[12] := WORD_TO_BYTE(左下悬挂伺服电流 AND 16#FF);
tmpDataSend[13] := WORD_TO_BYTE(SHR(左下悬挂伺服位置, 8));
tmpDataSend[14] := WORD_TO_BYTE(左下悬挂伺服位置 AND 16#FF);
tmpDataSend[15] := WORD_TO_BYTE(SHR(左下悬挂伺服速度, 8));
tmpDataSend[16] := WORD_TO_BYTE(左下悬挂伺服速度 AND 16#FF);
tmpDataSend[17] := WORD_TO_BYTE(SHR(左下悬挂伺服温度, 8));
tmpDataSend[18] := WORD_TO_BYTE(左下悬挂伺服温度 AND 16#FF);
tmpDataSend[19] := WORD_TO_BYTE(SHR(左下悬挂伺服报错码, 8));
tmpDataSend[20] := WORD_TO_BYTE(左下悬挂伺服报错码 AND 16#FF);
tmpDataSend[21] := 16#01;	//0-离线 1-在线

tmpDataSend[22] := WORD_TO_BYTE(SHR(右上悬挂伺服电流, 8));
tmpDataSend[23] := WORD_TO_BYTE(右上悬挂伺服电流 AND 16#FF);
tmpDataSend[24] := WORD_TO_BYTE(SHR(右上悬挂伺服位置, 8));
tmpDataSend[25] := WORD_TO_BYTE(右上悬挂伺服位置 AND 16#FF);
tmpDataSend[26] := WORD_TO_BYTE(SHR(右上悬挂伺服速度, 8));
tmpDataSend[27] := WORD_TO_BYTE(右上悬挂伺服速度 AND 16#FF);
tmpDataSend[28] := WORD_TO_BYTE(SHR(右上悬挂伺服温度, 8));
tmpDataSend[29] := WORD_TO_BYTE(右上悬挂伺服温度 AND 16#FF);
tmpDataSend[30] := WORD_TO_BYTE(SHR(右上悬挂伺服报错码, 8));
tmpDataSend[31] := WORD_TO_BYTE(右上悬挂伺服报错码 AND 16#FF);
tmpDataSend[32] := 16#01;	//0-离线 1-在线

tmpDataSend[33] := WORD_TO_BYTE(SHR(右下悬挂伺服电流, 8));
tmpDataSend[34] := WORD_TO_BYTE(右下悬挂伺服电流 AND 16#FF);
tmpDataSend[35] := WORD_TO_BYTE(SHR(右下悬挂伺服位置, 8));
tmpDataSend[36] := WORD_TO_BYTE(右下悬挂伺服位置 AND 16#FF);
tmpDataSend[37] := WORD_TO_BYTE(SHR(右下悬挂伺服速度, 8));
tmpDataSend[38] := WORD_TO_BYTE(右下悬挂伺服速度 AND 16#FF);
tmpDataSend[39] := WORD_TO_BYTE(SHR(右下悬挂伺服温度, 8));
tmpDataSend[40] := WORD_TO_BYTE(右下悬挂伺服温度 AND 16#FF);
tmpDataSend[41] := WORD_TO_BYTE(SHR(右下悬挂伺服报错码, 8));
tmpDataSend[42] := WORD_TO_BYTE(右下悬挂伺服报错码 AND 16#FF);
tmpDataSend[43] := 16#01;	//0-离线 1-在线

上传信息处理_4(定时时间:=T#1100MS, 数据域长度:=44, pInputData:=ADR(tmpDataSend[0]), 应答:=16#00, 序列号:=上传序列号, 主功能码:=16#04, 次功能码:=16#02);
END_METHOD

METHOD 轮速计数据上传
VAR_INPUT
END_VAR
VAR
	线速度: WORD;
	角速度: WORD;	
END_VAR
//轮速计数据 [0x04,0x0D]
线速度 := LREAL_TO_WORD((左下轮伺服参数.反馈速度 - 右下轮伺服参数.反馈速度) / 2 / 1000);
角速度 := LREAL_TO_WORD((右下轮伺服参数.反馈速度 + 左下轮伺服参数.反馈速度) / 1.6935 / 1000);

tmpDataSend[0] := 0;
tmpDataSend[1] := 0;
tmpDataSend[2] := WORD_TO_BYTE(SHR(线速度, 8));
tmpDataSend[3] := WORD_TO_BYTE(线速度 AND 16#FF);

tmpDataSend[4] := 0;
tmpDataSend[5] := 0;
tmpDataSend[6] := WORD_TO_BYTE(SHR(角速度, 8));
tmpDataSend[7] := WORD_TO_BYTE(角速度 AND 16#FF);

上传信息处理_7(定时时间:=T#20MS, 数据域长度:=8, pInputData:=ADR(tmpDataSend[0]), 应答:=16#02, 序列号:=上传序列号, 主功能码:=16#04, 次功能码:=16#0D);
END_METHOD

METHOD UPS数据上传
VAR_INPUT
END_VAR
VAR
	电池过程数据	: WORD;
END_VAR
// UPS数据[0x04,0x0F] 
// 报警状态码（9字节，byte[0~8]
tmpDataSend[0] := WORD_TO_BYTE(SHR(BMS映射数据[0], 8));
tmpDataSend[1] := WORD_TO_BYTE(BMS映射数据[0] AND 16#FF);
tmpDataSend[2] := WORD_TO_BYTE(SHR(BMS映射数据[1], 8));
tmpDataSend[3] := WORD_TO_BYTE(BMS映射数据[1] AND 16#FF);
tmpDataSend[4] := WORD_TO_BYTE(SHR(BMS映射数据[2], 8));
tmpDataSend[5] := WORD_TO_BYTE(BMS映射数据[2] AND 16#FF);
tmpDataSend[6] := WORD_TO_BYTE(SHR(BMS映射数据[3], 8));
tmpDataSend[7] := WORD_TO_BYTE(BMS映射数据[3] AND 16#FF);
tmpDataSend[8] := WORD_TO_BYTE(SHR(BMS映射数据[4], 8));
tmpDataSend[9] := WORD_TO_BYTE(BMS映射数据[4] AND 16#FF);

// 2. 电气参数
// 2.1 R相输入电压
电池过程数据 := LREAL_TO_WORD(R输入电压 * 10) ;  			// 转换为0.1V
tmpDataSend[10] := LREAL_TO_BYTE(SHR(电池过程数据, 8));
tmpDataSend[11] := WORD_TO_BYTE(电池过程数据 AND 16#FF);

// 2.2 S相输入电压
电池过程数据 := LREAL_TO_WORD(S输入电压 * 10) ;  			// 转换为0.1V
tmpDataSend[12] := LREAL_TO_BYTE(SHR(电池过程数据, 8));
tmpDataSend[13] := WORD_TO_BYTE(电池过程数据 AND 16#FF);

// 2.3 T相输入电压
电池过程数据 := LREAL_TO_WORD(T输入电压 * 10) ;  			// 转换为0.1V
tmpDataSend[14] := LREAL_TO_BYTE(SHR(电池过程数据, 8));
tmpDataSend[15] := WORD_TO_BYTE(电池过程数据 AND 16#FF);

// 2.4 输入频率电池未提供->(当前功率)
tmpDataSend[16] := LREAL_TO_BYTE(SHR(UPS映射数据[26], 8));
tmpDataSend[17] := WORD_TO_BYTE(UPS映射数据[26] AND 16#FF);

// 2.5 R相输出电压
tmpDataSend[18] := LREAL_TO_BYTE(SHR(UPS映射数据[9], 8));	// 转换为0.1V
tmpDataSend[19] := WORD_TO_BYTE(UPS映射数据[9] AND 16#FF);

// 2.6 S相输出电压
tmpDataSend[20] := LREAL_TO_BYTE(SHR(UPS映射数据[10], 8));// 转换为0.1V
tmpDataSend[21] := WORD_TO_BYTE(UPS映射数据[10] AND 16#FF);

// 2.7 T相输出电压
tmpDataSend[22] := LREAL_TO_BYTE(SHR(UPS映射数据[11], 8));// 转换为0.1V
tmpDataSend[23] := WORD_TO_BYTE(UPS映射数据[11] AND 16#FF);

// 2.8 输出频率
tmpDataSend[24] := LREAL_TO_BYTE(SHR(UPS映射数据[12], 8));// 转换为0.1V
tmpDataSend[25] := WORD_TO_BYTE(UPS映射数据[12] AND 16#FF);

// 2.9 R相输出电流
tmpDataSend[26] := LREAL_TO_BYTE(SHR(UPS映射数据[13], 8));
tmpDataSend[27] := WORD_TO_BYTE(UPS映射数据[13] AND 16#FF);

// 2.10 S相输出电流
tmpDataSend[28] := LREAL_TO_BYTE(SHR(UPS映射数据[14], 8));
tmpDataSend[29] := WORD_TO_BYTE(UPS映射数据[14] AND 16#FF);

// 2.11 T相输出电流
tmpDataSend[30] := LREAL_TO_BYTE(SHR(UPS映射数据[15], 8));
tmpDataSend[31] := WORD_TO_BYTE(UPS映射数据[15] AND 16#FF);

// 2.12 R相输出功率比率 
tmpDataSend[32] := LREAL_TO_BYTE(SHR(UPS映射数据[16], 8));
tmpDataSend[33] := WORD_TO_BYTE(UPS映射数据[16] AND 16#FF);

// 2.13 S相输出功率比率
tmpDataSend[34] := LREAL_TO_BYTE(SHR(UPS映射数据[17], 8));
tmpDataSend[35] := WORD_TO_BYTE(UPS映射数据[17] AND 16#FF);

// 2.14 T相输出功率比率
tmpDataSend[36] := LREAL_TO_BYTE(SHR(UPS映射数据[18], 8));
tmpDataSend[37] := WORD_TO_BYTE(UPS映射数据[18] AND 16#FF);

// 2.15 三相输出功率比率 
tmpDataSend[38] := LREAL_TO_BYTE(SHR(UPS映射数据[19], 8));
tmpDataSend[39] := WORD_TO_BYTE(UPS映射数据[19] AND 16#FF);

// 2.16 UPS状态字    
tmpDataSend[40] := LREAL_TO_BYTE(SHR(UPS映射数据[20], 8)); 
tmpDataSend[41] := WORD_TO_BYTE(UPS映射数据[20] AND 16#FF);

// 2.17 散热器温度1 
tmpDataSend[42] := LREAL_TO_BYTE(SHR(UPS映射数据[21], 8)); 
tmpDataSend[43] := WORD_TO_BYTE(UPS映射数据[21] AND 16#FF);

// 2.18 散热器温度2
tmpDataSend[44] := LREAL_TO_BYTE(SHR(UPS映射数据[22], 8)); 
tmpDataSend[45] := WORD_TO_BYTE(UPS映射数据[22] AND 16#FF); 

// 2.19 UPS温度
tmpDataSend[46] := LREAL_TO_BYTE(SHR(UPS映射数据[23], 8));
tmpDataSend[47] := WORD_TO_BYTE(UPS映射数据[23] AND 16#FF); 

// 3. UPS当前工作模式
tmpDataSend[48] := WORD_TO_BYTE(UPS映射数据[24]); //0x50-开机模式 0x53-待机模式 0x59-旁路模式 0x4C-线路模式 0x42-电池模式 0x46-故障模式 0x45-HE/ECO模式 0x43-转换器模式 0x44-关机模式 

tmpDataSend[49] := LREAL_TO_BYTE(SHR(UPS映射数据[25], 8));
tmpDataSend[50] := WORD_TO_BYTE(UPS映射数据[25] AND 16#FF); 

//4. 上传报文
上传信息处理_6(定时时间:=T#9980MS, 数据域长度:=51, pInputData:=ADR(tmpDataSend[0]), 应答:=16#00, 序列号:=上传序列号, 主功能码:=16#04, 次功能码:=16#0F);
END_METHOD

METHOD 超声波数据上传
VAR_INPUT
END_VAR
VAR
	边沿左上	: WORD;
	边沿左下	: WORD;
	边沿右上	: WORD;
	边沿右下	: WORD;
	超声波左1	: WORD;
	超声波左2	: WORD;
	超声波右1	: WORD;
	超声波右2	: WORD;
END_VAR
//超声波数据 [0x04,0x05]
边沿左上 := LREAL_TO_WORD(边沿检测1);
边沿左下 := LREAL_TO_WORD(边沿检测2);
边沿右上 := LREAL_TO_WORD(边沿检测3);
边沿右下 := LREAL_TO_WORD(边沿检测4);
超声波左1 := LREAL_TO_WORD(超声波检测左1);
超声波左2 := LREAL_TO_WORD(超声波检测左2);
超声波右1 := LREAL_TO_WORD(超声波检测右1);
超声波右2 := LREAL_TO_WORD(超声波检测右2);

tmpDataSend[0] := WORD_TO_BYTE(SHR(边沿左上, 8));
tmpDataSend[1] := WORD_TO_BYTE(边沿左上 AND 16#FF);
tmpDataSend[2] := WORD_TO_BYTE(SHR(边沿左下, 8));
tmpDataSend[3] := WORD_TO_BYTE(边沿左下 AND 16#FF);
tmpDataSend[4] := WORD_TO_BYTE(SHR(边沿右上, 8));
tmpDataSend[5] := WORD_TO_BYTE(边沿右上 AND 16#FF);
tmpDataSend[6] := WORD_TO_BYTE(SHR(边沿右下, 8));
tmpDataSend[7] := WORD_TO_BYTE(边沿右下 AND 16#FF);

tmpDataSend[8] := WORD_TO_BYTE(SHR(超声波左1, 8));
tmpDataSend[9] := WORD_TO_BYTE(超声波左1 AND 16#FF);
tmpDataSend[10] := WORD_TO_BYTE(SHR(超声波左2, 8));
tmpDataSend[11] := WORD_TO_BYTE(超声波左2 AND 16#FF);
tmpDataSend[12] := WORD_TO_BYTE(SHR(超声波右1, 8));
tmpDataSend[13] := WORD_TO_BYTE(超声波右1 AND 16#FF);
tmpDataSend[14] := WORD_TO_BYTE(SHR(超声波右2, 8));
tmpDataSend[15] := WORD_TO_BYTE(超声波右2 AND 16#FF);

上传信息处理_1(定时时间:=T#500MS, 数据域长度:=16, pInputData:=ADR(tmpDataSend[0]), 应答:=16#00, 序列号:=上传序列号, 主功能码:=16#04, 次功能码:=16#05);
END_METHOD

END_PROGRAM

// Device/Application/函数/SLAM通讯/校验功能块
FUNCTION_BLOCK 校验功能块
VAR_INPUT
	pData: POINTER TO BYTE;
	sizeNome: WORD;
END_VAR
VAR_OUTPUT
	sumCheck: BYTE;
END_VAR
VAR
	i: WORD;
END_VAR

sumCheck := 0;
FOR i:=1 TO sizeNome BY 1 DO	
	sumCheck := sumCheck + pData^;
	pData := pData + SIZEOF(BYTE);
END_FOR

END_FUNCTION_BLOCK

// Device/Application/函数/SLAM通讯/上传信息处理
FUNCTION_BLOCK 上传信息处理
VAR_INPUT
	定时时间: TIME := T#0S;
	数据域长度: BYTE := 0;
	pInputData: POINTER TO BYTE;
	应答: BYTE;
	主功能码: BYTE;
	次功能码: BYTE;
END_VAR
VAR_OUTPUT
END_VAR
VAR_IN_OUT
	序列号: WORD;
END_VAR
VAR
	tmpSize: BYTE;
	tmpData: ARRAY[0..200] OF BYTE;
	i: BYTE;
	校验功能块_0: 校验功能块;
	sumcheck: BYTE;
	tmpByte: POINTER TO BYTE;
	TON_0: TON;
	定时启动: BOOL;
END_VAR

///
TON_0(IN:=定时启动 , PT:=定时时间 , Q=> , ET=> );
IF NOT 定时启动  THEN
	定时启动 := 1;
END_IF

IF TON_0.Q OR 定时时间 = T#0S THEN
	定时启动 := 0;
	
	///////////////////////////////////////////////////数据处理
	tmpData[0] := 16#5A;
	tmpData[1] := 16#A5;
	tmpData[3] := WORD_TO_BYTE(SHR(序列号, 8));
	tmpData[4] := WORD_TO_BYTE(序列号);
	tmpData[5] := 主功能码;
	tmpData[6] := 次功能码;
	tmpData[7]:= 应答;
	tmpSize := 6 + 数据域长度;
	tmpData[2] := tmpSize+1;
	IF 数据域长度 <> 0 THEN
		FOR i:=1 TO 数据域长度  BY 1 DO		
			tmpData[7+i] :=pInputData^;
			pInputData := pInputData + SIZEOF(BYTE);
		END_FOR
	END_IF
	校验功能块_0(pData:=ADR(tmpData[0]), sizeNome:=tmpSize + 2 , sumCheck=>tmpData[7 + 数据域长度 +1] );
	tmpSize := tmpData[2] +2 ;
	///////////////////////////////////////////////////发送处理
	AryMove(In:=tmpData[0] , AryOut:=待发送缓存数组[待发送缓存数组长度] , Size:= tmpSize);
	待发送缓存数组长度 := 待发送缓存数组长度 + tmpSize;
	IF 主功能码 = 16#04 THEN
		IF 序列号 = 65534 THEN
			序列号 := 0;
		ELSE
			序列号 := 序列号 +1;
		END_IF
		  
	END_IF
END_IF

END_FUNCTION_BLOCK

// Device/Application/函数/SLAM通讯/上传信息处理_1
FUNCTION_BLOCK 上传信息处理_1

VAR_INPUT
	定时时间: TIME := T#0S;
	数据域长度: BYTE := 0;
	pInputData: POINTER TO BYTE;
	应答: BYTE;
END_VAR
VAR_IN_OUT
	序列号: WORD;
END_VAR
VAR_INPUT
	主功能码: BYTE;
	次功能码: BYTE;
END_VAR
VAR
	tmpSize: BYTE;
	tmpData: ARRAY[0..200] OF BYTE;
	i: BYTE;
	校验功能块_0: 校验功能块;
	sumcheck: BYTE;
	tmpByte: POINTER TO BYTE;
	TON_0: TON;
	定时启动: BOOL;
END_VAR

///
TON_0(IN:=定时启动 , PT:=定时时间 , Q=> , ET=> );
IF NOT 定时启动  THEN
	定时启动 := 1;
END_IF

IF TON_0.Q OR 定时时间 = T#0S THEN
	定时启动 := 0;
	
	///////////////////////////////////////////////////数据处理
	tmpData[0] := 16#5A;
	tmpData[1] := 16#A5;
	tmpData[3] := WORD_TO_BYTE(SHR(序列号, 8));
	tmpData[4] := WORD_TO_BYTE(序列号);
	tmpData[5] := 主功能码;
	tmpData[6] := 次功能码;
	tmpData[7]:= 应答;
	tmpSize := 6 + 数据域长度;
	tmpData[2] := tmpSize+1;
	IF 数据域长度 <> 0 THEN
		FOR i:=1 TO 数据域长度  BY 1 DO		
			tmpData[7+i] :=pInputData^;
			pInputData := pInputData + SIZEOF(BYTE);
		END_FOR
	END_IF
	校验功能块_0(pData:=ADR(tmpData[0]), sizeNome:=tmpSize + 2 , sumCheck=>tmpData[7 + 数据域长度 +1] );
	tmpSize := tmpData[2] +2 ;
	///////////////////////////////////////////////////发送处理
	AryMove(In:=tmpData[0] , AryOut:=业务通讯待发送缓存数组[业务通讯待发送缓存数组长度] , Size:= tmpSize);
	业务通讯待发送缓存数组长度 := 业务通讯待发送缓存数组长度 + tmpSize;
	IF 主功能码 = 16#04 THEN
		IF 序列号 = 65534 THEN
			序列号 := 0;
		ELSE
			序列号 := 序列号 +1;
		END_IF
		  
	END_IF
END_IF

END_FUNCTION_BLOCK

// Device/Application/SLAM业务通讯
PROGRAM SLAM业务通讯	
VAR
	作业控制编码 	: WORD;
	流程处理状态 	: INT := 100;
	清扫返回功能码 : BYTE;
	清扫返回状态 : BYTE;
	清扫作业流程处理 : 清扫作业流程;
	SktTCPSend_0: SktTCPSend;
	SktTCPRecv_0: SktTCPRecv;
	SktClose_0: SktClose;
	SktTCPGetStatus_0: SktTCPGetStatus;
	diConnectID: CONNECT_ID := 50;
	stServerAddress: ADDRESS;
	stConnectInfo: CONNECT_INFO;
	DataSend: ARRAY[0..1024] OF BYTE;
	DataRevice: ARRAY[0..1024] OF BYTE;
	status: WORD := 0;
	R_TRIG_0: R_TRIG;
	F_TRIG_0: F_TRIG;
	start_tcp_server: BOOL;
	SktTCPServer_0: SktTCPServer;
	CanWR: BOOL;
	HandleDataRevice: ARRAY[0..2048] OF BYTE;
	NumRevc: WORD := 0;
	tmpRevc: WORD := 0;
	i: WORD := 0;
	校验功能块_0: 校验功能块;
	sumcheck: BYTE;
	SendSize: WORD;
	bSend: BOOL;
	tmpDataSend: ARRAY[0..200] OF BYTE;
	接收序列号: WORD;
	初始化: BOOL;
	TON_0: TON;
	TON_2: TON;
	bCloseSocket: BOOL := 0;
	上传信息处理_0: 	上传信息处理_1;	
	上传信息处理_1:	上传信息处理_1;	
END_VAR

R_TRIG_0(CLK:=业务通讯复位, Q=> );
F_TRIG_0(CLK:=业务通讯复位 , Q=> );

TON_0(IN:=业务通讯自动重连 AND status = 255 , PT:=T#1S , Q=> , ET=> );
TON_2(IN:=SktClose_0.xExecute AND status = 4 , PT:=T#3S , Q=> , ET=> );
IF TON_2.Q THEN
	status := 1;
	SktClose_0(xExecute:=FALSE);		
	SktTCPGetStatus_0(xEnable:=FALSE);
	start_tcp_server := FALSE;	
	CanWR := 0;
	NumRevc :=0;
	业务通讯连接状态 := 0;
	bSend := 0;
	bCloseSocket := 0;
END_IF


IF F_TRIG_0.Q OR NOT 初始化 OR TON_0.Q THEN
	status := 1;
END_IF
IF   R_TRIG_0.Q  THEN 
	IF status=1 THEN
		status := 255;
	ELSIF status=2 THEN
		status := 255;
	ELSIF status=3 THEN
		status := 4;
	END_IF	
END_IF

SktTCPServer_0(
		xExecute:= start_tcp_server, 
		diConnectID:= diConnectID, 
		strLocalAddress:= stServerAddress, 
		xDone=> , 
		xBusy=> , 
		xError=> , 
		wErrorID=> , 
		stConnectInfo=> stConnectInfo);

SktClose_0(
		xExecute:= bCloseSocket, 
		diConnectID:=stConnectInfo.diConnectID ,
		xDone=> ,
		xBusy=> ,
		xError=> ,
		wErrorID=> );


CASE status OF
	1:
		业务通讯连接状态 := 0;
		stServerAddress.strIPAddr := '0.0.0.0';
		stServerAddress.uiPort := 8002;
		start_tcp_server := TRUE;
		status := 2;
		CanWR := 0;
		bCloseSocket := 0;
	2:		
		IF SktTCPServer_0.xDone THEN
			status := 3;
			JMP RUN_RND;			
		ELSIF SktTCPServer_0.xError THEN		
			IF SktTCPServer_0.wErrorID = 21 THEN
				IF diConnectID <100 THEN
					diConnectID := diConnectID +1;
				ELSE
					diConnectID := 50;
				END_IF
				
			ELSE
				status := 255;
			END_IF
					
			JMP RUN_RND;
		END_IF
	3:
		CanWR := 0;
		SktTCPGetStatus_0(
			xEnable:= TRUE, 
			diConnectID:= stConnectInfo.diConnectID, 
			xDone=> , 
			xBusy=> , 
			xError=> , 
			wErrorID=> , 
			eStatus=> , 
			stConnectInfo=> );
		IF SktTCPGetStatus_0.xError THEN
			status := 4;
			业务通讯连接状态 := 0;
			JMP RUN_RND;
		ELSIF SktTCPGetStatus_0.eStatus <> CmpHCTCPIP.TCP_STATUS.TCP_ESTABLISHED THEN
			status := 4;
			业务通讯连接状态 := 0;
			JMP RUN_RND;
			;
		ELSE
			业务通讯连接状态 := 1;
			CanWR := 1;
		END_IF
	4:
		bCloseSocket := 1;
		IF SktClose_0.xDone THEN
			status := 255;
			JMP RUN_RND;
		END_IF
		CanWR :=0;
	255:
		bCloseSocket := 0;		
		SktTCPGetStatus_0(xEnable:=FALSE);
		start_tcp_server := FALSE;	
		CanWR := 0;
		NumRevc :=0;
		业务通讯连接状态 := 0;
		bSend := 0;
ELSE
	;
END_CASE

SktTCPRecv_0(
	xEnable:= CanWR, 
	diConnectID:= stConnectInfo.diConnectID, 
	abyData:= DataRevice[0], 
	uiDataSize:= 0, 
	xDone=> , 
	xBusy=> , 
	xError=> , 
	wErrorID=> , 
	xReady=> , 
	uiCount=> );
IF SktTCPRecv_0.xError THEN
	status := 4;
	JMP RUN_RND;
ELSIF SktTCPRecv_0.xDone AND NOT(SktTCPRecv_0.xError) THEN
	status := 255;
	JMP RUN_RND;
ELSE
	IF SktTCPRecv_0.xReady THEN
		tmpRevc := 0;
		IF (2048-NumRevc) < SktTCPRecv_0.uiCount THEN
			tmpRevc := SktTCPRecv_0.uiCount - (2048-NumRevc);					
		END_IF
		AryMove(In:=DataRevice[0] , AryOut:=HandleDataRevice[NumRevc] , Size:=SktTCPRecv_0.uiCount - tmpRevc );	
		NumRevc := NumRevc + SktTCPRecv_0.uiCount - tmpRevc;
	END_IF	
END_IF
tmpRevc := 0;

IF NumRevc >= 7 AND NumRevc < 2048 THEN
    FOR i := 0 TO NumRevc - 1 BY 1 DO
        IF HandleDataRevice[i] = 16#5A THEN
            IF (NumRevc - i) >= 7 THEN
                IF HandleDataRevice[i + 1] = 16#A5 THEN
                    IF (i + HandleDataRevice[i + 2] + 2) <= NumRevc THEN
                        校验功能块_0(pData := ADR(HandleDataRevice[i]), sizeNome := HandleDataRevice[i + 2] + 1, sumCheck => sumcheck);
                        IF HandleDataRevice[HandleDataRevice[i + 2] + 1 + i] = sumcheck THEN
                            CASE HandleDataRevice[i + 5] OF
                                16#02: //作业状态设置
									IF HandleDataRevice[i+6] = 16#05 THEN
										光伏板离地高度 := WORD_TO_INT(SHL(BYTE_TO_WORD(HandleDataRevice[i+9]), 8) OR HandleDataRevice[i+10]);
										光伏板角度 := WORD_TO_INT(SHL(BYTE_TO_WORD(HandleDataRevice[i+11]), 8) OR HandleDataRevice[i+12]);
										IF HandleDataRevice[i+13]=16#55 THEN
											光伏板方向 := -1.0;
										ELSIF HandleDataRevice[i+13]=16#AA THEN
											光伏板方向 := 1.0;
										END_IF
										接收序列号 := SHL(BYTE_TO_WORD( HandleDataRevice[i+3]), 8) OR HandleDataRevice[i+4];
										作业控制编码 := SHL(BYTE_TO_WORD(HandleDataRevice[i+7]), 8) OR HandleDataRevice[i+8];
										CASE 作业控制编码 OF
											16#0101 : //系统初始化
												流程处理状态 := 0;
												tmpDataSend[0] := 16#01;
												tmpDataSend[1] := 16#00;
												上传信息处理_0(定时时间:=T#0MS, 数据域长度:=2, pInputData:=ADR(tmpDataSend[0]), 应答:=16#00, 序列号:=接收序列号, 主功能码:=16#02, 次功能码:=16#05);
											16#0202 : //清扫待命状态
												流程处理状态 := 10;
												tmpDataSend[0] := 16#02;
												tmpDataSend[1] := 16#00;
												上传信息处理_0(定时时间:=T#0MS, 数据域长度:=2, pInputData:=ADR(tmpDataSend[0]), 应答:=16#00, 序列号:=接收序列号, 主功能码:=16#02, 次功能码:=16#05);
											16#0303 : //清扫准备状态
												流程处理状态 := 20;
												tmpDataSend[0] := 16#03;
												tmpDataSend[1] := 16#00;
												上传信息处理_0(定时时间:=T#0MS, 数据域长度:=2, pInputData:=ADR(tmpDataSend[0]), 应答:=16#00, 序列号:=接收序列号, 主功能码:=16#02, 次功能码:=16#05);
											16#0404 : //清扫暂停状态
												流程处理状态 := 30;
												tmpDataSend[0] := 16#04;
												tmpDataSend[1] := 16#00;
												上传信息处理_0(定时时间:=T#0MS, 数据域长度:=2, pInputData:=ADR(tmpDataSend[0]), 应答:=16#00, 序列号:=接收序列号, 主功能码:=16#02, 次功能码:=16#05);
											16#0505 : //行走复位状态
												流程处理状态 := 40;
												tmpDataSend[0] := 16#05;
												tmpDataSend[1] := 16#00;
												上传信息处理_0(定时时间:=T#0MS, 数据域长度:=2, pInputData:=ADR(tmpDataSend[0]), 应答:=16#00, 序列号:=接收序列号, 主功能码:=16#02, 次功能码:=16#05);
											16#0B0B : //急停状态
												流程处理状态 := 1;
											16#0C0C : //进入现场操作模式
												流程处理状态 := 1;
											16#0D0D : //退出现场操作模式
												流程处理状态 := 1;
										END_CASE
                                    END_IF
									
// 									IF HandleDataRevice[i+6] = 16#06 THEN
// 										上装数据上传();
//                                     END_IF
                            END_CASE
                            i := i + HandleDataRevice[i + 2] + 1;
                            tmpRevc := i + 1;
                        END_IF
                    ELSE
                        JMP
                        RUN_ENDFOR;
                    END_IF
                ELSE
                    tmpRevc := tmpRevc + 1;
                END_IF
            ELSE
                JMP
                RUN_ENDFOR;
            END_IF
        ELSE
            tmpRevc := tmpRevc + 1;
        END_IF;
    END_FOR
END_IF

清扫作业流程处理(作业状态:=流程处理状态, 离地高度:=光伏板离地高度, 光伏板角度:=光伏板角度, 离车间距:=光伏板离底盘中心距离, 清扫方向:=光伏板方向, 返回功能码=>清扫返回功能码, 返回状态=>清扫返回状态);
IF 清扫返回状态 = 16#05 THEN
	流程处理状态 := 100;
	tmpDataSend[0] := 清扫返回功能码;
	tmpDataSend[1] := 清扫返回状态;
	上传信息处理_1(定时时间:=T#0MS, 数据域长度:=2, pInputData:=ADR(tmpDataSend[0]), 应答:=16#00, 序列号:=接收序列号, 主功能码:=16#02, 次功能码:=16#05);
END_IF

RUN_ENDFOR:
IF tmpRevc > 0 THEN
	ArySHR(InOut:=HandleDataRevice[0] , Size:=2048 , Num:=tmpRevc );
	NumRevc := NumRevc - tmpRevc;
END_IF

IF 业务通讯待发送缓存数组长度 >0 AND bSend = 0 THEN
	SendSize := 业务通讯待发送缓存数组长度;
	AryMove(In:=业务通讯待发送缓存数组[0] , AryOut:=DataSend[0] , Size:= SendSize);
	业务通讯待发送缓存数组长度 :=0;
	bSend := 1;
END_IF

SktTCPSend_0(
	xExecute:= bSend, 
	diConnectID:= stConnectInfo.diConnectID, 
	abyData:= DataSend[0], 
	uiDataSize:= SendSize, 
	uiTimeOut:= 500, 
	xDone=> , 
	xBusy=> , 
	xError=> , 
	wErrorID=> );
IF SktTCPSend_0.xError THEN
	status := 4;
	JMP RUN_RND;
ELSIF SktTCPSend_0.xDone THEN
	bSend := 0; //发送完毕
	SendSize := 0;
END_IF
		
RUN_RND:

//SLAM通讯不上 := NOT SLAM连接状态;
IF NOT 初始化 THEN
	初始化 :=1;
// 	// 每 20 s 刷新一次（其实只在第一次扫描时执行一次）
//     FOR i := 1 TO 16 DO
//         ProbeTemp[i] := BYTE(50 + i MOD 20);   // 50..69 → 0..19 ℃
//     END_FOR
END_IF

METHOD 上装数据上传
VAR_INPUT
END_VAR
VAR
	机械臂一轴电流	: WORD;
	机械臂一轴速度	: WORD;
	机械臂一轴位置	: WORD;
	机械臂一轴温度	: WORD;
	机械臂一轴报错码	: WORD;
	
	机械臂二轴电流	: WORD;
	机械臂二轴速度	: WORD;
	机械臂二轴位置	: WORD;
	机械臂二轴温度	: WORD;
	机械臂二轴报错码	: WORD;
	
	机械臂三轴电流	: WORD;
	机械臂三轴速度	: WORD;
	机械臂三轴位置	: WORD;
	机械臂三轴温度	: WORD;
	机械臂三轴报错码	: WORD;

	机械臂四轴电流	: WORD;
	机械臂四轴速度	: WORD;
	机械臂四轴位置	: WORD;
	机械臂四轴温度	: WORD;
	机械臂四轴报错码	: WORD;
	
	伸缩轴伺服电流	: WORD;
	伸缩轴伺服速度	: WORD;
	伸缩轴伺服位置	: WORD;
	伸缩轴伺服温度	: WORD;
	伸缩轴伺服报错码	: WORD;
	
	上卷扬伺服电流	: WORD;
	上卷扬伺服速度	: WORD;
	上卷扬伺服位置	: WORD;
	上卷扬伺服温度	: WORD;
	上卷扬伺服报错码	: WORD;
	
	下卷扬伺服电流	: WORD;
	下卷扬伺服速度	: WORD;
	下卷扬伺服位置	: WORD;
	下卷扬伺服温度	: WORD;
	下卷扬伺服报错码	: WORD;
	
	滚刷伺服电流		: WORD;
	滚刷伺服速度		: WORD;
	滚刷伺服温度		: WORD;
	滚刷伺服报错码	: WORD;
	
	左前测距超声波数据	: WORD;
	右前测距超声波数据	: WORD;
	左后测距超声波数据	: WORD;
	右后测距超声波数据	: WORD;
	左前边沿超声波数据	: WORD;
	右前边沿超声波数据	: WORD;
	左后边沿超声波数据	: WORD;
	右后边沿超声波数据	: WORD;
	
	机械臂空间X		: WORD;
	机械臂空间Y		: WORD;
	机械臂空间Z		: WORD;
	机械臂空间B		: WORD;
	底盘俯仰角		: WORD;
	底盘横滚角		: WORD;
	机械臂运行状态	: WORD;
	机械臂报错码		: WORD;
END_VAR
//上装数据 [0x02,0x06]
机械臂一轴电流 := LREAL_TO_WORD(左上轮伺服参数.反馈电流);
机械臂一轴速度 := LREAL_TO_WORD(37);
机械臂一轴位置 := LREAL_TO_WORD(0);
机械臂一轴温度 := LREAL_TO_WORD(37);
机械臂一轴报错码 := LREAL_TO_WORD(0);

机械臂二轴电流 := LREAL_TO_WORD(左下轮伺服参数.反馈电流);
机械臂二轴速度 := LREAL_TO_WORD(37);
机械臂二轴位置 := LREAL_TO_WORD(0);
机械臂二轴温度 := LREAL_TO_WORD(37);
机械臂二轴报错码 := LREAL_TO_WORD(0);

机械臂三轴电流 := LREAL_TO_WORD(右上轮伺服参数.反馈电流);
机械臂三轴速度 := LREAL_TO_WORD(37);
机械臂三轴位置 := LREAL_TO_WORD(0);
机械臂三轴温度 := LREAL_TO_WORD(37);
机械臂三轴报错码 := LREAL_TO_WORD(0);

机械臂四轴电流 := LREAL_TO_WORD(右下轮伺服参数.反馈电流);
机械臂四轴速度 := LREAL_TO_WORD(37);
机械臂四轴位置 := LREAL_TO_WORD(0);
机械臂四轴温度 := LREAL_TO_WORD(37);
机械臂四轴报错码 := LREAL_TO_WORD(0);

伸缩轴伺服电流 := LREAL_TO_WORD(伸缩轴伺服参数.反馈电流);
伸缩轴伺服速度 := LREAL_TO_WORD(37);
伸缩轴伺服位置 := LREAL_TO_WORD(0);
伸缩轴伺服温度 := LREAL_TO_WORD(37);
伸缩轴伺服报错码 := LREAL_TO_WORD(0);

上卷扬伺服电流 := LREAL_TO_WORD(右下轮伺服参数.反馈电流);
上卷扬伺服速度 := LREAL_TO_WORD(37);
上卷扬伺服位置 := LREAL_TO_WORD(0);
上卷扬伺服温度 := LREAL_TO_WORD(37);
上卷扬伺服报错码 := LREAL_TO_WORD(0);

下卷扬伺服电流 := LREAL_TO_WORD(右下轮伺服参数.反馈电流);
下卷扬伺服速度 := LREAL_TO_WORD(37);
下卷扬伺服位置 := LREAL_TO_WORD(0);
下卷扬伺服温度 := LREAL_TO_WORD(37);
下卷扬伺服报错码 := LREAL_TO_WORD(0);

滚刷伺服电流 := LREAL_TO_WORD(右下轮伺服参数.反馈电流);
滚刷伺服速度 := LREAL_TO_WORD(37);
滚刷伺服温度 := LREAL_TO_WORD(0);
滚刷伺服报错码 := LREAL_TO_WORD(37);

左前测距超声波数据 := LREAL_TO_WORD(0);
右前测距超声波数据 := LREAL_TO_WORD(37);
左后测距超声波数据 := LREAL_TO_WORD(0);
右后测距超声波数据 := LREAL_TO_WORD(37);
左前边沿超声波数据 := LREAL_TO_WORD(0);
右前边沿超声波数据 := LREAL_TO_WORD(0);
左后边沿超声波数据 := LREAL_TO_WORD(0);
右后边沿超声波数据 := LREAL_TO_WORD(0);

机械臂空间X := LREAL_TO_WORD(右下轮伺服参数.反馈电流);
机械臂空间Y := LREAL_TO_WORD(37);
机械臂空间Z := LREAL_TO_WORD(0);
机械臂空间B := LREAL_TO_WORD(37);
底盘俯仰角 := LREAL_TO_WORD(0);
底盘横滚角 := LREAL_TO_WORD(0);

tmpDataSend[0] := WORD_TO_BYTE(SHR(机械臂一轴电流, 8));
tmpDataSend[1] := WORD_TO_BYTE(机械臂一轴电流 AND 16#FF);
tmpDataSend[2] := WORD_TO_BYTE(SHR(机械臂一轴速度, 8));
tmpDataSend[3] := WORD_TO_BYTE(机械臂一轴速度 AND 16#FF);
tmpDataSend[4] := WORD_TO_BYTE(SHR(机械臂一轴位置, 8));
tmpDataSend[5] := WORD_TO_BYTE(机械臂一轴位置 AND 16#FF);
tmpDataSend[6] := WORD_TO_BYTE(SHR(机械臂一轴温度, 8));
tmpDataSend[7] := WORD_TO_BYTE(机械臂一轴温度 AND 16#FF);
tmpDataSend[8] := WORD_TO_BYTE(SHR(机械臂一轴报错码, 8));
tmpDataSend[5] := WORD_TO_BYTE(机械臂一轴报错码 AND 16#FF);
tmpDataSend[10] := 16#01;	//0-离线 1-在线

tmpDataSend[11] := WORD_TO_BYTE(SHR(机械臂二轴电流, 8));
tmpDataSend[12] := WORD_TO_BYTE(机械臂二轴电流 AND 16#FF);
tmpDataSend[13] := WORD_TO_BYTE(SHR(机械臂二轴速度, 8));
tmpDataSend[14] := WORD_TO_BYTE(机械臂二轴速度 AND 16#FF);
tmpDataSend[15] := WORD_TO_BYTE(SHR(机械臂二轴位置, 8));
tmpDataSend[16] := WORD_TO_BYTE(机械臂二轴位置 AND 16#FF);
tmpDataSend[17] := WORD_TO_BYTE(SHR(机械臂二轴温度, 8));
tmpDataSend[18] := WORD_TO_BYTE(机械臂二轴温度 AND 16#FF);
tmpDataSend[19] := WORD_TO_BYTE(SHR(机械臂二轴报错码, 8));
tmpDataSend[20] := WORD_TO_BYTE(机械臂二轴报错码 AND 16#FF);
tmpDataSend[21] := 16#01;	//0-离线 1-在线

tmpDataSend[22] := WORD_TO_BYTE(SHR(机械臂三轴电流, 8));
tmpDataSend[23] := WORD_TO_BYTE(机械臂三轴电流 AND 16#FF);
tmpDataSend[24] := WORD_TO_BYTE(SHR(机械臂三轴速度, 8));
tmpDataSend[25] := WORD_TO_BYTE(机械臂三轴速度 AND 16#FF);
tmpDataSend[26] := WORD_TO_BYTE(SHR(机械臂三轴位置, 8));
tmpDataSend[27] := WORD_TO_BYTE(机械臂三轴位置 AND 16#FF);
tmpDataSend[28] := WORD_TO_BYTE(SHR(机械臂三轴温度, 8));
tmpDataSend[29] := WORD_TO_BYTE(机械臂三轴温度 AND 16#FF);
tmpDataSend[30] := WORD_TO_BYTE(SHR(机械臂三轴报错码, 8));
tmpDataSend[31] := WORD_TO_BYTE(机械臂三轴报错码 AND 16#FF);
tmpDataSend[32] := 16#01;	//0-离线 1-在线

tmpDataSend[33] := WORD_TO_BYTE(SHR(机械臂四轴电流, 8));
tmpDataSend[34] := WORD_TO_BYTE(机械臂四轴电流 AND 16#FF);
tmpDataSend[35] := WORD_TO_BYTE(SHR(机械臂四轴速度, 8));
tmpDataSend[36] := WORD_TO_BYTE(机械臂四轴速度 AND 16#FF);
tmpDataSend[37] := WORD_TO_BYTE(SHR(机械臂四轴位置, 8));
tmpDataSend[38] := WORD_TO_BYTE(机械臂四轴位置 AND 16#FF);
tmpDataSend[39] := WORD_TO_BYTE(SHR(机械臂四轴温度, 8));
tmpDataSend[40] := WORD_TO_BYTE(机械臂四轴温度 AND 16#FF);
tmpDataSend[41] := WORD_TO_BYTE(SHR(机械臂四轴报错码, 8));
tmpDataSend[42] := WORD_TO_BYTE(机械臂四轴报错码 AND 16#FF);
tmpDataSend[43] := 16#01;	//0-离线 1-在线

tmpDataSend[44] := WORD_TO_BYTE(SHR(伸缩轴伺服电流, 8));
tmpDataSend[45] := WORD_TO_BYTE(伸缩轴伺服电流 AND 16#FF);
tmpDataSend[46] := WORD_TO_BYTE(SHR(伸缩轴伺服速度, 8));
tmpDataSend[47] := WORD_TO_BYTE(伸缩轴伺服速度 AND 16#FF);
tmpDataSend[48] := WORD_TO_BYTE(SHR(伸缩轴伺服位置, 8));
tmpDataSend[49] := WORD_TO_BYTE(伸缩轴伺服位置 AND 16#FF);
tmpDataSend[50] := WORD_TO_BYTE(SHR(伸缩轴伺服温度, 8));
tmpDataSend[51] := WORD_TO_BYTE(伸缩轴伺服温度 AND 16#FF);
tmpDataSend[52] := WORD_TO_BYTE(SHR(伸缩轴伺服报错码, 8));
tmpDataSend[53] := WORD_TO_BYTE(伸缩轴伺服报错码 AND 16#FF);
tmpDataSend[54] := 16#01;	//0-离线 1-在线

tmpDataSend[55] := WORD_TO_BYTE(SHR(上卷扬伺服电流, 8));
tmpDataSend[56] := WORD_TO_BYTE(上卷扬伺服电流 AND 16#FF);
tmpDataSend[57] := WORD_TO_BYTE(SHR(上卷扬伺服速度, 8));
tmpDataSend[58] := WORD_TO_BYTE(上卷扬伺服速度 AND 16#FF);
tmpDataSend[59] := WORD_TO_BYTE(SHR(上卷扬伺服位置, 8));
tmpDataSend[60] := WORD_TO_BYTE(上卷扬伺服位置 AND 16#FF);
tmpDataSend[61] := WORD_TO_BYTE(SHR(上卷扬伺服温度, 8));
tmpDataSend[62] := WORD_TO_BYTE(上卷扬伺服温度 AND 16#FF);
tmpDataSend[63] := WORD_TO_BYTE(SHR(上卷扬伺服报错码, 8));
tmpDataSend[64] := WORD_TO_BYTE(上卷扬伺服报错码 AND 16#FF);
tmpDataSend[65] := 16#01;	//0-离线 1-在线

